(* CODESYS project 车床桁架_RECOVERED_2024-04-15T14-33-14.project
   CompiledLibraryCompatibilityVersion: LeadSysStudio V3.5 SP15 Patch 4
   Title: 车床桁架

Project tree, tasks and I/O mapping:
  Device : SC5-C0A4, Leadshine Technology Co., Ltd., order no. 504001, version 3.5.15.40
    application Application
      libraries: Standard, * (System)
      task MainTask (cyclic, interval t#20ms, priority 1) calls PLC_PRG, 气缸, Public_Prog, OP1001, OP1002
      task EtherCAT_Master_Leadshine_A (cyclic, interval 4000 µs, priority 0) calls EtherCAT_Master_Leadshine_A.EtherCAT_Task, Servo_Ctrol
      program 回原 [LD]
      FunctionBlock/
        function block FB102_ClockPuls [LD]
        program Public_Prog [LD]: SystemVar
        function block FB_CylinderDouble [ST]
        function block FB_CylinderSingle [ST]
      global variables HMI
      global variables I_List
      global variables Alarm
      Symbols
      data type CYLINDER_REF
      global variables 气缸_STRUCT
      program OP1002 [LD]: 辅助流程
      global variables System
      program 气缸 [LD]
      program Servo_Ctrol [LD]
      global variables Publics
      interface ITF
      global variables PersistentVars
      program PLC_PRG [LD]
      program OP1001 [LD]
      global variables O_Lisk
    Device Diagnose
    Network Configuration
      LocalBus Config
    Resource Usage
    LocalBus_Master_Module : LocalBusR1 Master, Leadshine Technology Co., Ltd., version 3.5.15.40
      SC0032N1 : SC0032N1, Leadshine Technology Co., Ltd., version 3.5.15.40
          settings: 位置号 = 1
          unmapped channels: OUTPUT_0, OUTPUT_1, OUTPUT_2, OUTPUT_3
      SC3200 : SC3200, Leadshine Technology Co., Ltd., version 3.5.15.40
          settings: 位置号 = 0
          unmapped channels: INPUT_0, INPUT_1, INPUT_2, INPUT_3
    Modbus_Slave_RS232_COM : Modbus Slave RS232 COM, Leadshine Technology Co., Ltd., version 3.5.15.40
        settings: Vendor.Baudrate = 115200
    SoftMotion General Axis Pool
    EtherCAT_Master_Leadshine_A : EtherCAT Master SoftMotion, 3S - Smart Software Solutions GmbH, version 3.5.16.30
        settings: NetworkName = 'ecat'; SelectNetworkByName = TRUE
      L6N_2 : L6N(COE), Leadshine Technology Co.,Ltd., order no. L6N, version Revision=16#00000001
          settings: DC sync0 cycletime = 4000; DC sync1 cycletime = 4000; Number of SDO = 6; Homing method.Index = 16#6098; Homing method.Subindex = 16#00; Homing method.Value = 35; Homing method.Size = 8; Homing method.AbortIfError = FALSE; Homing method.JumpToLine = FALSE; Homing method.Line = 0; Homing method.CompleteAccess = FALSE; Homing velocity (fast).Index = 16#6099; Homing velocity (fast).Subindex = 16#01; Homing velocity (fast).Value = 6103261; Homing velocity (fast).Size = 32; Homing velocity (fast).AbortIfError = FALSE; Homing velocity (fast).JumpToLine = FALSE; Homing velocity (fast).Line = 0; Homing velocity (fast).CompleteAccess = FALSE; Homing velocity (slow).Index = 16#6099; Homing velocity (slow).Subindex = 16#02; Homing velocity (slow).Value = 1220652; Homing velocity (slow).Size = 32; Homing velocity (slow).AbortIfError = FALSE; Homing velocity (slow).JumpToLine = FALSE; Homing velocity (slow).Line = 0; Homing velocity (slow).CompleteAccess = FALSE; Homing acceleration.Index = 16#609A; Homing acceleration.Subindex = 16#00; Homing acceleration.Value = 61032615; Homing acceleration.Size = 32; Homing acceleration.AbortIfError = FALSE; Homing acceleration.JumpToLine = FALSE; Homing acceleration.Line = 0; Homing acceleration.CompleteAccess = FALSE; Homing offset.Index = 16#607C; Homing offset.Subindex = 16#00; Homing offset.Value = 0; Homing offset.Size = 32; Homing offset.AbortIfError = FALSE;
            Homing offset.JumpToLine = FALSE; Homing offset.Line = 0; Homing offset.CompleteAccess = FALSE
          unmapped channels: Control word, Profile target position, Touch Probe Function, Last error code, Status word, Modes of operation display, Position loop error, Actual motor torque, Actual motor position, Touch Probe Status, Touch probe pos1 pos value, Digital inputs
        Axis_2 : Axis, 3S - Smart Software Solutions GmbH, order no. 0, version 4.6.1.0
            settings: wDriveID = 2; bVirtual = TRUE; dwRatioTechUnitsDenom = 610326149; iRatioTechUnitsNum = 1000; fSWMaxVelocity = 1000; fSWMaxAcceleration = 10000; fSWMaxDeceleration = 10000; fSWMaxJerk = 100000; 一圈脉冲数 = 8388608; 工作台一圈的位移 = 109.955741; 电子齿轮比分子 = 8; 电子齿轮比分母 = 1; ScalingIncs = 8388608; ScalingMotorTurns2 = 8; AdrOffset_8010 = 28; BitOffset_8010 = 0; BitLength_8010 = 16; Address_8010 = '%QW14'; Type_8010 = 'UINT'; AddressPointer_8010 = ADR(%QW14); AdrOffset_8020 = 32; BitOffset_8020 = 0; BitLength_8020 = 32; Address_8020 = '%QD8'; Type_8020 = 'DINT'; AddressPointer_8020 = ADR(%QD8); AdrOffset_8030 = 4294967295; BitOffset_8030 = 0; BitLength_8030 = 32; Address_8030 = ''; Type_8030 = 'DINT'; AddressPointer_8030 = 0; AdrOffset_8040 = 4294967295; BitOffset_8040 = 0; BitLength_8040 = 16; Address_8040 = ''; Type_8040 = 'INT'; AddressPointer_8040 = 0; AdrOffset_8050 = 4294967295; BitOffset_8050 = 0;
              BitLength_8050 = 8; Address_8050 = ''; Type_8050 = 'SINT'; AddressPointer_8050 = 0; AdrOffset_8060 = 36; BitOffset_8060 = 0; BitLength_8060 = 16; Address_8060 = '%QW18'; Type_8060 = 'UINT'; AddressPointer_8060 = ADR(%QW18); AdrOffset_8070 = 4294967295; BitOffset_8070 = 0; BitLength_8070 = 0; Address_8070 = ''; Type_8070 = ''; AddressPointer_8070 = 0; AdrOffset_8080 = 4294967295; BitOffset_8080 = 0; BitLength_8080 = 16; Address_8080 = ''; Type_8080 = 'INT'; AddressPointer_8080 = 0; AdrOffset_8090 = 4294967295; BitOffset_8090 = 0; BitLength_8090 = 0; Address_8090 = ''; Type_8090 = ''; AddressPointer_8090 = 0; AdrOffset_8510 = 70; BitOffset_8510 = 0; BitLength_8510 = 16; Address_8510 = '%IW35'; Type_8510 = 'UINT'; AddressPointer_8510 = ADR(%IW35); AdrOffset_8520 = 84; BitOffset_8520 = 0; BitLength_8520 = 32; Address_8520 = '%ID21'; Type_8520 = 'DINT'; AddressPointer_8520 = ADR(%ID21);
              AdrOffset_8530 = 4294967295; BitOffset_8530 = 0; BitLength_8530 = 0; Address_8530 = ''; Type_8530 = ''; AddressPointer_8530 = 0; AdrOffset_8540 = 80; BitOffset_8540 = 0; BitLength_8540 = 16; Address_8540 = '%IW40'; Type_8540 = 'INT'; AddressPointer_8540 = ADR(%IW40); AdrOffset_8550 = 72; BitOffset_8550 = 0; BitLength_8550 = 8; Address_8550 = '%IB72'; Type_8550 = 'SINT'; AddressPointer_8550 = ADR(%IB72); AdrOffset_8560 = 96; BitOffset_8560 = 0; BitLength_8560 = 32; Address_8560 = '%ID24'; Type_8560 = 'UDINT'; AddressPointer_8560 = ADR(%ID24); AdrOffset_8570 = 88; BitOffset_8570 = 0; BitLength_8570 = 16; Address_8570 = '%IW44'; Type_8570 = 'UINT'; AddressPointer_8570 = ADR(%IW44); AdrOffset_8580 = 92; BitOffset_8580 = 0; BitLength_8580 = 32; Address_8580 = '%ID23'; Type_8580 = 'DINT'; AddressPointer_8580 = ADR(%ID23); AdrOffset_8590 = 4294967295; BitOffset_8590 = 0; BitLength_8590 = 0; Address_8590 = '';
              Type_8590 = ''; AddressPointer_8590 = 0; AdrOffset_8600 = 4294967295; BitOffset_8600 = 0; BitLength_8600 = 0; Address_8600 = ''; Type_8600 = ''; AddressPointer_8600 = 0; AdrOffset_8600 = 4294967295; BitOffset_8600 = 0; BitLength_8600 = 0; Address_8610 = ''; Type_8610 = ''; AddressPointer_8610 = 0; AdrOffset_8620 = 76; BitOffset_8620 = 0; BitLength_8620 = 32; Address_8620 = '%ID19'; Type_8620 = 'DINT'; AddressPointer_8620 = ADR(%ID19)
      L6N_3 : L6N(COE), Leadshine Technology Co.,Ltd., order no. L6N, version Revision=16#00000001
          settings: DC sync0 cycletime = 4000; DC sync1 cycletime = 4000; Number of SDO = 6; Homing method.Index = 16#6098; Homing method.Subindex = 16#00; Homing method.Value = 35; Homing method.Size = 8; Homing method.AbortIfError = FALSE; Homing method.JumpToLine = FALSE; Homing method.Line = 0; Homing method.CompleteAccess = FALSE; Homing velocity (fast).Index = 16#6099; Homing velocity (fast).Subindex = 16#01; Homing velocity (fast).Value = 26701769; Homing velocity (fast).Size = 32; Homing velocity (fast).AbortIfError = FALSE; Homing velocity (fast).JumpToLine = FALSE; Homing velocity (fast).Line = 0; Homing velocity (fast).CompleteAccess = FALSE; Homing velocity (slow).Index = 16#6099; Homing velocity (slow).Subindex = 16#02; Homing velocity (slow).Value = 5340354; Homing velocity (slow).Size = 32; Homing velocity (slow).AbortIfError = FALSE; Homing velocity (slow).JumpToLine = FALSE; Homing velocity (slow).Line = 0; Homing velocity (slow).CompleteAccess = FALSE; Homing acceleration.Index = 16#609A; Homing acceleration.Subindex = 16#00; Homing acceleration.Value = 267017690; Homing acceleration.Size = 32; Homing acceleration.AbortIfError = FALSE; Homing acceleration.JumpToLine = FALSE; Homing acceleration.Line = 0; Homing acceleration.CompleteAccess = FALSE; Homing offset.Index = 16#607C; Homing offset.Subindex = 16#00; Homing offset.Value = 0; Homing offset.Size = 32; Homing offset.AbortIfError = FALSE;
            Homing offset.JumpToLine = FALSE; Homing offset.Line = 0; Homing offset.CompleteAccess = FALSE
          unmapped channels: Control word, Profile target position, Touch Probe Function, Last error code, Status word, Modes of operation display, Position loop error, Actual motor torque, Actual motor position, Touch Probe Status, Touch probe pos1 pos value, Digital inputs
        Axis_3 : Axis, 3S - Smart Software Solutions GmbH, order no. 0, version 4.6.1.0
            settings: wDriveID = 3; bVirtual = TRUE; dwRatioTechUnitsDenom = 26701769; iRatioTechUnitsNum = 10; fSWMaxVelocity = 1000; fSWMaxAcceleration = 10000; fSWMaxDeceleration = 10000; fSWMaxJerk = 100000; 一圈脉冲数 = 8388608; 工作台一圈的位移 = 109.955741; 电子齿轮比分子 = 35; 电子齿轮比分母 = 1; ScalingIncs = 8388608; ScalingMotorTurns2 = 35; AdrOffset_8010 = 40; BitOffset_8010 = 0; BitLength_8010 = 16; Address_8010 = '%QW20'; Type_8010 = 'UINT'; AddressPointer_8010 = ADR(%QW20); AdrOffset_8020 = 44; BitOffset_8020 = 0; BitLength_8020 = 32; Address_8020 = '%QD11'; Type_8020 = 'DINT'; AddressPointer_8020 = ADR(%QD11); AdrOffset_8030 = 4294967295; BitOffset_8030 = 0; BitLength_8030 = 32; Address_8030 = ''; Type_8030 = 'DINT'; AddressPointer_8030 = 0; AdrOffset_8040 = 4294967295; BitOffset_8040 = 0; BitLength_8040 = 16; Address_8040 = ''; Type_8040 = 'INT'; AddressPointer_8040 = 0; AdrOffset_8050 = 4294967295; BitOffset_8050 = 0;
              BitLength_8050 = 8; Address_8050 = ''; Type_8050 = 'SINT'; AddressPointer_8050 = 0; AdrOffset_8060 = 48; BitOffset_8060 = 0; BitLength_8060 = 16; Address_8060 = '%QW24'; Type_8060 = 'UINT'; AddressPointer_8060 = ADR(%QW24); AdrOffset_8070 = 4294967295; BitOffset_8070 = 0; BitLength_8070 = 0; Address_8070 = ''; Type_8070 = ''; AddressPointer_8070 = 0; AdrOffset_8080 = 4294967295; BitOffset_8080 = 0; BitLength_8080 = 16; Address_8080 = ''; Type_8080 = 'INT'; AddressPointer_8080 = 0; AdrOffset_8090 = 4294967295; BitOffset_8090 = 0; BitLength_8090 = 0; Address_8090 = ''; Type_8090 = ''; AddressPointer_8090 = 0; AdrOffset_8510 = 102; BitOffset_8510 = 0; BitLength_8510 = 16; Address_8510 = '%IW51'; Type_8510 = 'UINT'; AddressPointer_8510 = ADR(%IW51); AdrOffset_8520 = 116; BitOffset_8520 = 0; BitLength_8520 = 32; Address_8520 = '%ID29'; Type_8520 = 'DINT'; AddressPointer_8520 = ADR(%ID29);
              AdrOffset_8530 = 4294967295; BitOffset_8530 = 0; BitLength_8530 = 0; Address_8530 = ''; Type_8530 = ''; AddressPointer_8530 = 0; AdrOffset_8540 = 112; BitOffset_8540 = 0; BitLength_8540 = 16; Address_8540 = '%IW56'; Type_8540 = 'INT'; AddressPointer_8540 = ADR(%IW56); AdrOffset_8550 = 104; BitOffset_8550 = 0; BitLength_8550 = 8; Address_8550 = '%IB104'; Type_8550 = 'SINT'; AddressPointer_8550 = ADR(%IB104); AdrOffset_8560 = 128; BitOffset_8560 = 0; BitLength_8560 = 32; Address_8560 = '%ID32'; Type_8560 = 'UDINT'; AddressPointer_8560 = ADR(%ID32); AdrOffset_8570 = 120; BitOffset_8570 = 0; BitLength_8570 = 16; Address_8570 = '%IW60'; Type_8570 = 'UINT'; AddressPointer_8570 = ADR(%IW60); AdrOffset_8580 = 124; BitOffset_8580 = 0; BitLength_8580 = 32; Address_8580 = '%ID31'; Type_8580 = 'DINT'; AddressPointer_8580 = ADR(%ID31); AdrOffset_8590 = 4294967295; BitOffset_8590 = 0; BitLength_8590 = 0; Address_8590 = '';
              Type_8590 = ''; AddressPointer_8590 = 0; AdrOffset_8600 = 4294967295; BitOffset_8600 = 0; BitLength_8600 = 0; Address_8600 = ''; Type_8600 = ''; AddressPointer_8600 = 0; AdrOffset_8600 = 4294967295; BitOffset_8600 = 0; BitLength_8600 = 0; Address_8610 = ''; Type_8610 = ''; AddressPointer_8610 = 0; AdrOffset_8620 = 108; BitOffset_8620 = 0; BitLength_8620 = 32; Address_8620 = '%ID27'; Type_8620 = 'DINT'; AddressPointer_8620 = ADR(%ID27)
      L6N_1 : L6N(COE), Leadshine Technology Co.,Ltd., order no. L6N, version Revision=16#00000001
          settings: DC sync0 cycletime = 4000; DC sync1 cycletime = 4000; Number of SDO = 6; Homing method.Index = 16#6098; Homing method.Subindex = 16#00; Homing method.Value = 35; Homing method.Size = 8; Homing method.AbortIfError = FALSE; Homing method.JumpToLine = FALSE; Homing method.Line = 0; Homing method.CompleteAccess = FALSE; Homing velocity (fast).Index = 16#6099; Homing velocity (fast).Subindex = 16#01; Homing velocity (fast).Value = 16777216; Homing velocity (fast).Size = 32; Homing velocity (fast).AbortIfError = FALSE; Homing velocity (fast).JumpToLine = FALSE; Homing velocity (fast).Line = 0; Homing velocity (fast).CompleteAccess = FALSE; Homing velocity (slow).Index = 16#6099; Homing velocity (slow).Subindex = 16#02; Homing velocity (slow).Value = 3355443; Homing velocity (slow).Size = 32; Homing velocity (slow).AbortIfError = FALSE; Homing velocity (slow).JumpToLine = FALSE; Homing velocity (slow).Line = 0; Homing velocity (slow).CompleteAccess = FALSE; Homing acceleration.Index = 16#609A; Homing acceleration.Subindex = 16#00; Homing acceleration.Value = 167772160; Homing acceleration.Size = 32; Homing acceleration.AbortIfError = FALSE; Homing acceleration.JumpToLine = FALSE; Homing acceleration.Line = 0; Homing acceleration.CompleteAccess = FALSE; Homing offset.Index = 16#607C; Homing offset.Subindex = 16#00; Homing offset.Value = 0; Homing offset.Size = 32; Homing offset.AbortIfError = FALSE;
            Homing offset.JumpToLine = FALSE; Homing offset.Line = 0; Homing offset.CompleteAccess = FALSE
          unmapped channels: Control word, Profile target position, Touch Probe Function, Last error code, Status word, Modes of operation display, Position loop error, Actual motor torque, Actual motor position, Touch Probe Status, Touch probe pos1 pos value, Digital inputs
        Axis_1 : Axis, 3S - Smart Software Solutions GmbH, order no. 0, version 4.6.1.0
            settings: bVirtual = TRUE; dwRatioTechUnitsDenom = 8388608; iRatioTechUnitsNum = 5; fSWMaxVelocity = 1000; fSWMaxAcceleration = 10000; fSWMaxDeceleration = 10000; fSWMaxJerk = 100000; 一圈脉冲数 = 8388608; 工作台一圈的位移 = 5; 电子齿轮比分子 = 1; 电子齿轮比分母 = 1; ScalingIncs = 8388608; AdrOffset_8010 = 16; BitOffset_8010 = 0; BitLength_8010 = 16; Address_8010 = '%QW8'; Type_8010 = 'UINT'; AddressPointer_8010 = ADR(%QW8); AdrOffset_8020 = 20; BitOffset_8020 = 0; BitLength_8020 = 32; Address_8020 = '%QD5'; Type_8020 = 'DINT'; AddressPointer_8020 = ADR(%QD5); AdrOffset_8030 = 4294967295; BitOffset_8030 = 0; BitLength_8030 = 32; Address_8030 = ''; Type_8030 = 'DINT'; AddressPointer_8030 = 0; AdrOffset_8040 = 4294967295; BitOffset_8040 = 0; BitLength_8040 = 16; Address_8040 = ''; Type_8040 = 'INT'; AddressPointer_8040 = 0; AdrOffset_8050 = 4294967295; BitOffset_8050 = 0; BitLength_8050 = 8; Address_8050 = '';
              Type_8050 = 'SINT'; AddressPointer_8050 = 0; AdrOffset_8060 = 24; BitOffset_8060 = 0; BitLength_8060 = 16; Address_8060 = '%QW12'; Type_8060 = 'UINT'; AddressPointer_8060 = ADR(%QW12); AdrOffset_8070 = 4294967295; BitOffset_8070 = 0; BitLength_8070 = 0; Address_8070 = ''; Type_8070 = ''; AddressPointer_8070 = 0; AdrOffset_8080 = 4294967295; BitOffset_8080 = 0; BitLength_8080 = 16; Address_8080 = ''; Type_8080 = 'INT'; AddressPointer_8080 = 0; AdrOffset_8090 = 4294967295; BitOffset_8090 = 0; BitLength_8090 = 0; Address_8090 = ''; Type_8090 = ''; AddressPointer_8090 = 0; AdrOffset_8510 = 38; BitOffset_8510 = 0; BitLength_8510 = 16; Address_8510 = '%IW19'; Type_8510 = 'UINT'; AddressPointer_8510 = ADR(%IW19); AdrOffset_8520 = 52; BitOffset_8520 = 0; BitLength_8520 = 32; Address_8520 = '%ID13'; Type_8520 = 'DINT'; AddressPointer_8520 = ADR(%ID13); AdrOffset_8530 = 4294967295; BitOffset_8530 = 0;
              BitLength_8530 = 0; Address_8530 = ''; Type_8530 = ''; AddressPointer_8530 = 0; AdrOffset_8540 = 48; BitOffset_8540 = 0; BitLength_8540 = 16; Address_8540 = '%IW24'; Type_8540 = 'INT'; AddressPointer_8540 = ADR(%IW24); AdrOffset_8550 = 40; BitOffset_8550 = 0; BitLength_8550 = 8; Address_8550 = '%IB40'; Type_8550 = 'SINT'; AddressPointer_8550 = ADR(%IB40); AdrOffset_8560 = 64; BitOffset_8560 = 0; BitLength_8560 = 32; Address_8560 = '%ID16'; Type_8560 = 'UDINT'; AddressPointer_8560 = ADR(%ID16); AdrOffset_8570 = 56; BitOffset_8570 = 0; BitLength_8570 = 16; Address_8570 = '%IW28'; Type_8570 = 'UINT'; AddressPointer_8570 = ADR(%IW28); AdrOffset_8580 = 60; BitOffset_8580 = 0; BitLength_8580 = 32; Address_8580 = '%ID15'; Type_8580 = 'DINT'; AddressPointer_8580 = ADR(%ID15); AdrOffset_8590 = 4294967295; BitOffset_8590 = 0; BitLength_8590 = 0; Address_8590 = ''; Type_8590 = ''; AddressPointer_8590 = 0;
              AdrOffset_8600 = 4294967295; BitOffset_8600 = 0; BitLength_8600 = 0; Address_8600 = ''; Type_8600 = ''; AddressPointer_8600 = 0; AdrOffset_8600 = 4294967295; BitOffset_8600 = 0; BitLength_8600 = 0; Address_8610 = ''; Type_8610 = ''; AddressPointer_8610 = 0; AdrOffset_8620 = 44; BitOffset_8620 = 0; BitLength_8620 = 32; Address_8620 = '%ID11'; Type_8620 = 'DINT'; AddressPointer_8620 = ADR(%ID11)
      L6N : L6N(COE), Leadshine Technology Co.,Ltd., order no. L6N, version Revision=16#00000001
          settings: DC sync0 cycletime = 4000; DC enable = 1; DC sync0 enable = 1; DC sync0 shift time = 0; DC sync1 cycletime = 4000; DC sync1 enable = 0; DC sync1 factor = 'x 1'; DC sync1 shift time = 0; Number of SDO = 6; Homing method.Index = 16#6098; Homing method.Subindex = 16#00; Homing method.Value = 35; Homing method.Size = 8; Homing method.AbortIfError = FALSE; Homing method.JumpToLine = FALSE; Homing method.Line = 0; Homing method.CompleteAccess = FALSE; Homing velocity (fast).Index = 16#6099; Homing velocity (fast).Subindex = 16#01; Homing velocity (fast).Value = 20971520; Homing velocity (fast).Size = 32; Homing velocity (fast).AbortIfError = FALSE; Homing velocity (fast).JumpToLine = FALSE; Homing velocity (fast).Line = 0; Homing velocity (fast).CompleteAccess = FALSE; Homing velocity (slow).Index = 16#6099; Homing velocity (slow).Subindex = 16#02; Homing velocity (slow).Value = 4194304; Homing velocity (slow).Size = 32; Homing velocity (slow).AbortIfError = FALSE; Homing velocity (slow).JumpToLine = FALSE; Homing velocity (slow).Line = 0; Homing velocity (slow).CompleteAccess = FALSE; Homing acceleration.Index = 16#609A; Homing acceleration.Subindex = 16#00; Homing acceleration.Value = 209715200; Homing acceleration.Size = 32; Homing acceleration.AbortIfError = FALSE; Homing acceleration.JumpToLine = FALSE; Homing acceleration.Line = 0;
            Homing acceleration.CompleteAccess = FALSE; Homing offset.Index = 16#607C; Homing offset.Subindex = 16#00; Homing offset.Value = 0; Homing offset.Size = 32; Homing offset.AbortIfError = FALSE; Homing offset.JumpToLine = FALSE; Homing offset.Line = 0; Homing offset.CompleteAccess = FALSE
          unmapped channels: Control word, Profile target position, Touch Probe Function, Last error code, Status word, Modes of operation display, Position loop error, Actual motor torque, Actual motor position, Touch Probe Status, Touch probe pos1 pos value, Digital inputs
        Axis : Axis, 3S - Smart Software Solutions GmbH, order no. 0, version 4.6.1.0
            settings: wDriveID = 0; bVirtual = TRUE; dwRatioTechUnitsDenom = 2097152; fSWMaxVelocity = 1000; fSWMaxAcceleration = 10000; fSWMaxDeceleration = 10000; fSWMaxJerk = 100000; 一圈脉冲数 = 8388608; 工作台一圈的位移 = 4; 电子齿轮比分子 = 1; 电子齿轮比分母 = 1; ScalingIncs = 8388608; AdrOffset_8010 = 4; BitOffset_8010 = 0; BitLength_8010 = 16; Address_8010 = '%QW2'; Type_8010 = 'UINT'; AddressPointer_8010 = ADR(%QW2); AdrOffset_8020 = 8; BitOffset_8020 = 0; BitLength_8020 = 32; Address_8020 = '%QD2'; Type_8020 = 'DINT'; AddressPointer_8020 = ADR(%QD2); AdrOffset_8030 = 4294967295; BitOffset_8030 = 0; BitLength_8030 = 32; Address_8030 = ''; Type_8030 = 'DINT'; AddressPointer_8030 = 0; AdrOffset_8040 = 4294967295; BitOffset_8040 = 0; BitLength_8040 = 16; Address_8040 = ''; Type_8040 = 'INT'; AddressPointer_8040 = 0; AdrOffset_8050 = 4294967295; BitOffset_8050 = 0; BitLength_8050 = 8; Address_8050 = '';
              Type_8050 = 'SINT'; AddressPointer_8050 = 0; AdrOffset_8060 = 12; BitOffset_8060 = 0; BitLength_8060 = 16; Address_8060 = '%QW6'; Type_8060 = 'UINT'; AddressPointer_8060 = ADR(%QW6); AdrOffset_8070 = 4294967295; BitOffset_8070 = 0; BitLength_8070 = 0; Address_8070 = ''; Type_8070 = ''; AddressPointer_8070 = 0; AdrOffset_8080 = 4294967295; BitOffset_8080 = 0; BitLength_8080 = 16; Address_8080 = ''; Type_8080 = 'INT'; AddressPointer_8080 = 0; AdrOffset_8090 = 4294967295; BitOffset_8090 = 0; BitLength_8090 = 0; Address_8090 = ''; Type_8090 = ''; AddressPointer_8090 = 0; AdrOffset_8510 = 6; BitOffset_8510 = 0; BitLength_8510 = 16; Address_8510 = '%IW3'; Type_8510 = 'UINT'; AddressPointer_8510 = ADR(%IW3); AdrOffset_8520 = 20; BitOffset_8520 = 0; BitLength_8520 = 32; Address_8520 = '%ID5'; Type_8520 = 'DINT'; AddressPointer_8520 = ADR(%ID5); AdrOffset_8530 = 4294967295; BitOffset_8530 = 0;
              BitLength_8530 = 0; Address_8530 = ''; Type_8530 = ''; AddressPointer_8530 = 0; AdrOffset_8540 = 16; BitOffset_8540 = 0; BitLength_8540 = 16; Address_8540 = '%IW8'; Type_8540 = 'INT'; AddressPointer_8540 = ADR(%IW8); AdrOffset_8550 = 8; BitOffset_8550 = 0; BitLength_8550 = 8; Address_8550 = '%IB8'; Type_8550 = 'SINT'; AddressPointer_8550 = ADR(%IB8); AdrOffset_8560 = 32; BitOffset_8560 = 0; BitLength_8560 = 32; Address_8560 = '%ID8'; Type_8560 = 'UDINT'; AddressPointer_8560 = ADR(%ID8); AdrOffset_8570 = 24; BitOffset_8570 = 0; BitLength_8570 = 16; Address_8570 = '%IW12'; Type_8570 = 'UINT'; AddressPointer_8570 = ADR(%IW12); AdrOffset_8580 = 28; BitOffset_8580 = 0; BitLength_8580 = 32; Address_8580 = '%ID7'; Type_8580 = 'DINT'; AddressPointer_8580 = ADR(%ID7); AdrOffset_8590 = 4294967295; BitOffset_8590 = 0; BitLength_8590 = 0; Address_8590 = ''; Type_8590 = ''; AddressPointer_8590 = 0;
              AdrOffset_8600 = 4294967295; BitOffset_8600 = 0; BitLength_8600 = 0; Address_8600 = ''; Type_8600 = ''; AddressPointer_8600 = 0; AdrOffset_8600 = 4294967295; BitOffset_8600 = 0; BitLength_8600 = 0; Address_8610 = ''; Type_8610 = ''; AddressPointer_8610 = 0; AdrOffset_8620 = 12; BitOffset_8620 = 0; BitLength_8620 = 32; Address_8620 = '%ID3'; Type_8620 = 'DINT'; AddressPointer_8620 = ADR(%ID3)
*)

// Device/Application/CYLINDER_REF
TYPE CYLINDER_REF :
STRUCT
	///初始化时返回原位控制
	xInit: BOOL;
	///自动控制,变为TRUE时，执行到位控制，变为FALSE时执行原位控制
	xAutoCmd: BOOL;
	///到位标志,处于原位状态
	xIsBack: BOOL;
	///到位标志,处于到位状态	
	xIsFront: BOOL;
END_STRUCT
END_TYPE

// Device/Application/HMI
{attribute 'qualified_only'}
VAR_GLOBAL
END_VAR
VAR_GLOBAL
	报警复位 AT %MX0.0: BOOL;
END_VAR
VAR_GLOBAL RETAIN PERSISTENT
	上料推出气缸原位延时 AT %MW1002: WORD := 10;
	上料推出气缸到位延时 AT %MW1003: WORD := 10;
END_VAR
VAR_GLOBAL
	上料顶起气缸_ON_UP AT %MX0.3: BOOL;
END_VAR
VAR_GLOBAL RETAIN PERSISTENT
	上料顶起气缸原位延时 AT %MW1000: WORD := 10;
	上料顶起气缸到位位延时 AT %MW1001: WORD := 10;
END_VAR
VAR_GLOBAL
	上料气动振动筛_ON_UP AT %MX0.6: BOOL;
	X轴失能 AT %MX0.7: BOOL;
	Z2轴失能 AT %MX1.0: BOOL;
	Z1轴失能 AT %MX1.1: BOOL;
	Y轴失能 AT %MX1.2: BOOL;
	X轴_CCW AT %MX1.3: BOOL;
	X轴_CW AT %MX1.4: BOOL;
	Y轴_CCW AT %MX1.5: BOOL;
	Y轴_CW AT %MX0.5: BOOL;
	Z1轴_CCW AT %MX0.4: BOOL;
	Z1轴_CW AT %MX1.6: BOOL;
	Z2轴_CCW AT %MX0.2: BOOL;
	Z2轴_CW AT %MX0.1: BOOL;
	上料推出气缸_ON_UP AT %MX1.7: BOOL;
END_VAR
VAR_GLOBAL RETAIN PERSISTENT
	X轴手动速度 AT %MD1000: REAL := 20;
	Z1轴手动速度 AT %MD1002: REAL := 20;
	Y轴手动速度 AT %MD1001: REAL := 20;
	Z2轴手动速度 AT %MD1003: REAL := 20;
	X轴手动减速度: REAL := 1000;
	X轴手动加速度: REAL := 1000;
	Y轴手动加速度: REAL := 1000;
	Y轴手动减速度: REAL := 1000;
	Z1轴手动减速度: REAL := 1000;
	Z1轴手动加速度: REAL := 1000;
	Z2轴手动减速度: REAL := 1000;
	Z2轴手动加速度: REAL := 1000;
END_VAR
VAR_GLOBAL
	X轴错误代码: DWORD;
	X状态_未使能 AT %MX2.4: BOOL;
	X状态_报错 AT %MX2.5: BOOL;
	X状态_停止中 AT %MX2.6: BOOL;
	X状态_准备好 AT %MX2.7: BOOL;
	X状态_点位运动 AT %MX3.0: BOOL;
	X状态_连续运动: BOOL;
	X状态_同步运动: BOOL;
	X状态_回零中: BOOL;
	X状态_恒速运动 AT %MX3.1: BOOL;
	X状态_加速中 AT %MX3.2: BOOL;
	X状态_减速中 AT %MX3.3: BOOL;
	X状态_超过软限制 AT %MX3.4: BOOL;
	Y轴错误代码: DWORD;
	Y状态_未使能 AT %MX3.5: BOOL;
	Y状态_报错 AT %MX3.6: BOOL;
	Y状态_停止中 AT %MX3.7: BOOL;
	Y状态_准备好 AT %MX4.0: BOOL;
	Y状态_点位运动 AT %MX4.1: BOOL;
	Y状态_连续运动: BOOL;
	Y状态_同步运动: BOOL;
	Y状态_回零中: BOOL;
	Y状态_恒速运动 AT %MX4.2: BOOL;
	Y状态_加速中 AT %MX4.3: BOOL;
	Y状态_减速中 AT %MX4.4: BOOL;
	Y状态_超过软限制 AT %MX4.5: BOOL;
	Z1轴错误代码: DWORD;
	Z1状态_未使能 AT %MX4.6: BOOL;
	Z1状态_报错 AT %MX4.7: BOOL;
	Z1状态_停止中 AT %MX5.0: BOOL;
	Z1状态_准备好 AT %MX5.1: BOOL;
	Z1状态_点位运动 AT %MX5.2: BOOL;
	Z1状态_连续运动: BOOL;
	Z1状态_同步运动: BOOL;
	Z1状态_回零中: BOOL;
	Z1状态_恒速运动 AT %MX5.3: BOOL;
	Z1状态_加速中 AT %MX5.4: BOOL;
	Z1状态_减速中 AT %MX5.5: BOOL;
	Z1状态_超过软限制 AT %MX5.6: BOOL;
	Z2轴错误代码: DWORD;
	Z2状态_未使能 AT %MX5.7: BOOL;
	Z2状态_报错 AT %mx6.0: BOOL;
	Z2状态_停止中 AT %mx6.1: BOOL;
	Z2状态_准备好 AT %MX6.7: BOOL;
	Z2状态_点位运动 AT %MX6.2: BOOL;
	Z2状态_连续运动: BOOL;
	Z2状态_同步运动: BOOL;
	Z2状态_回零中: BOOL;
	Z2状态_恒速运动 AT %MX6.3: BOOL;
	Z2状态_加速中 AT %MX6.4: BOOL;
	Z2状态_减速中 AT %MX6.5: BOOL;
	Z2状态_超过软限制 AT %MX6.6: BOOL;
	上料气爪_ON_UP AT %MX2.3: BOOL;
	开门气缸_ON_UP AT %MX2.2: BOOL;
	翻转气缸_ON_UP AT %MX2.1: BOOL;
	下料气爪_ON_UP AT %MX2.0: BOOL;
END_VAR
VAR_GLOBAL RETAIN PERSISTENT
	点位P0 AT %MD2000: ARRAY[0..3] OF REAL;
	点位P1 AT %MD2004: ARRAY[0..3] OF REAL;
END_VAR

VAR_GLOBAL
	Y轴当前位置 AT %MD1005: REAL;
	Z2轴当前位置 AT %MD1007: REAL;
	Z1轴当前位置 AT %MD1006: REAL;
	X轴当前位置 AT %MD1004: REAL;
	Z2当前速度: REAL;
	Z1当前速度: REAL;
	Y轴当前速度: REAL;
	X轴当前速度: REAL;
END_VAR
VAR_GLOBAL RETAIN PERSISTENT
	上料气爪原位延时 AT %MW1004: WORD := 10;
	上料气爪到位延时 AT %MW1005: WORD := 10;
	下料气爪到位延时 AT %MW1006: WORD := 10;
	下料气爪原位延时 AT %MW1007: WORD := 10;
	翻转气爪到位延时 AT %MW1008: WORD := 10;
	翻转气爪原位延时 AT %MW1009: WORD := 10;
	开门气缸原位延时 AT %MW1010: WORD := 50;
	开门气缸到位延时 AT %MW1011: WORD := 50;
	点位P9 AT %MD2036: ARRAY[0..3] OF REAL;
	点位P8 AT %MD2032: ARRAY[0..3] OF REAL;
	点位P7 AT %MD2028: ARRAY[0..3] OF REAL;
	点位P6 AT %MD2024: ARRAY[0..3] OF REAL;
	点位P5 AT %MD2020: ARRAY[0..3] OF REAL;
	点位P4 AT %MD2016: ARRAY[0..3] OF REAL;
	点位P3 AT %MD2012: ARRAY[0..3] OF REAL;
	点位P2 AT %MD2008: ARRAY[0..3] OF REAL;
	点位P10 AT %MD2040: ARRAY[0..3] OF REAL;
END_VAR

// Device/Application/I_List
{attribute 'qualified_only'}
VAR_GLOBAL
	// 上料传送带到位确认
	X0 AT %IX0.0: BOOL;
	// 紧急停止
	X1 AT %IX0.1: BOOL;
	// 推出气缸原位
	X2 AT %IX0.2: BOOL;
	// 推出气缸动作位
	X3 AT %IX0.3: BOOL;
	// 顶起气缸原位
	X4 AT %IX0.4: BOOL;
	// 顶起气缸动作位
	X5 AT %IX0.5: BOOL;
	// 上料气爪原位
	X6 AT %IX0.6: BOOL;
	// 上料气爪动作位
	X7 AT %IX0.7: BOOL;
	// 下料气爪原位
	X10 AT %IX1.0: BOOL;
	// 下料气爪动作位
	X11 AT %IX1.1: BOOL;
	// 翻转气缸原位
	X12 AT %IX1.2: BOOL;
	// 翻转气缸动作位
	X13 AT %IX1.3: BOOL;
	// 开门气缸原位
	X14 AT %IX1.4: BOOL;
	// 开门气缸动作位
	X15 AT %IX1.5: BOOL;
	// 启动按钮
	X16 AT %IX1.6: BOOL;
	// 停止按钮
	X17 AT %IX1.7: BOOL;
	// 复位按钮
	X20 AT %IX2.0: BOOL;
	// 手自动按钮ON为自动
	X21 AT %IX2.1: BOOL;
	// 下料确认
	X22 AT %IX2.2: BOOL;
	// 联机卡盘夹紧
	X23 AT %IX2.3: BOOL;
	// 联机启动
	X24 AT %IX2.4: BOOL;
	// 联机停止
	X25 AT %IX2.5: BOOL;
	// 联机故障
	X26 AT %IX2.6: BOOL;
	// 联机X轴零点
	X27 AT %IX2.7: BOOL;
	// 联机Z轴零点
	X30 AT %IX3.0: BOOL;
	X31 AT %IX3.1: BOOL;
	X32 AT %IX3.2: BOOL;
	X33 AT %IX3.3: BOOL;
	X34 AT %IX3.4: BOOL;
	X35 AT %IX3.5: BOOL;
	X36 AT %IX3.6: BOOL;
	X37 AT %IX3.7: BOOL;
END_VAR

// Device/Application/Alarm
{attribute 'qualified_only'}
VAR_GLOBAL
END_VAR
VAR_GLOBAL
	设备急停 AT %MX100.0: BOOL;
	推出气缸手自动不一致报警 AT %MX100.1: BOOL;
	推出气缸原位报警 AT %MX100.2: BOOL;
	推出气缸到位报警 AT %MX100.3: BOOL;
	顶起气缸手自动不一致报警 AT %MX100.4: BOOL;
	顶起气缸原位报警 AT %MX100.5: BOOL;
	顶起气缸到位报警 AT %MX100.6: BOOL;
	上料气爪手自动不一致报警 AT %MX100.7: BOOL;
	上料气爪原位报警 AT %MX101.0: BOOL;
	上料气爪到位报警 AT %MX101.1: BOOL;
	下料气爪手自动不一致报警 AT %MX101.2: BOOL;
	下料气爪原位报警 AT %MX101.3: BOOL;
	下料气爪到位报警 AT %MX101.4: BOOL;
	翻转气缸手自动不一致报警 AT %MX101.5: BOOL;
	翻转气缸原位报警 AT %MX101.6: BOOL;
	翻转气缸到位报警 AT %MX101.7: BOOL;
	开门气缸手自动不一致报警 AT %MX102.0: BOOL;
	开门气缸原位报警 AT %MX102.1: BOOL;
	开门气缸到位报警 AT %MX102.2: BOOL;
END_VAR

// Device/Application/气缸_STRUCT
{attribute 'qualified_only'}
VAR_GLOBAL
	上料推出气缸: CYLINDER_REF;
	上料顶起气缸: CYLINDER_REF;
	上料振动筛: CYLINDER_REF;
	开门气缸: CYLINDER_REF;
	翻转气缸: CYLINDER_REF;
	上料气爪: CYLINDER_REF;
	下料气爪: CYLINDER_REF;
END_VAR

// Device/Application/System
{attribute 'qualified_only'}
VAR_GLOBAL
	// 上电扫描一周期
FirstScan    :BOOL;
// 常ON
AlwaysTRUE   : BOOL;
// 常OFF
AlwaysFALSE  : BOOL;
// 0.1S周期脉冲
Clock_10Hz    :BOOL;
// 0.2S周期脉冲
Clock_5Hz    :BOOL;
// 0.5S周期脉冲
Clock_2Hz    :BOOL;
// 1S周期脉冲
Clock_1Hz    :BOOL;
// 2S周期脉冲
Clock_HalfHz :BOOL;
END_VAR

// Device/Application/Publics
{attribute 'qualified_only'}
VAR_GLOBAL
	// 调试使用常ON
CYGIA_ON   :BOOL;
// 调试使用常OFF
CYGIA_OFF  :BOOL;
	启动上升: BOOL;
	警报: BOOL;
	暂停: BOOL;
	EMG: BOOL;
	X定位数据: REAL;
	Y定位数据: REAL;
	Z1定位数据: REAL;
	Z2定位数据: REAL;
	Z2加速度: REAL;
	Z1加速度: REAL;
END_VAR
VAR_GLOBAL RETAIN PERSISTENT
	Y加速度: REAL;
	X加速度: REAL;
	Z2减速度: REAL;
	Z1减速度: REAL;
	Y减速度: REAL;
	X减速度: REAL;
	Z2自动速度: REAL;
	Z1自动速度: REAL;
	Y自动速度: REAL;
	X自动速度: REAL;
END_VAR
VAR_GLOBAL
	Z2轴完成: BOOL;
	Z1轴完成: BOOL;
	Y轴完成: BOOL;
	X轴完成: BOOL;
	Z2轴启动: BOOL;
	Z1轴启动: BOOL;
	Y轴启动: BOOL;
	X轴启动: BOOL;
END_VAR

// Device/Application/PersistentVars
{attribute 'qualified_only'}
VAR_GLOBAL PERSISTENT RETAIN
	// 生成持久变量的实例路径
	HMI.上料推出气缸原位延时: WORD := WORD#10;
	// 生成持久变量的实例路径
	HMI.上料推出气缸到位延时: WORD := WORD#10;
	// 生成持久变量的实例路径
	HMI.上料顶起气缸原位延时: WORD := WORD#10;
	// 生成持久变量的实例路径
	HMI.上料顶起气缸到位位延时: WORD := WORD#10;
	// 生成持久变量的实例路径
	HMI.X轴手动速度: REAL := 20.0;
	// 生成持久变量的实例路径
	HMI.Z1轴手动速度: REAL := 20.0;
	// 生成持久变量的实例路径
	HMI.Y轴手动速度: REAL := 20.0;
	// 生成持久变量的实例路径
	HMI.Z2轴手动速度: REAL := 20.0;
	// 生成持久变量的实例路径
	HMI.X轴手动减速度: REAL := 1000.0;
	// 生成持久变量的实例路径
	HMI.X轴手动加速度: REAL := 1000.0;
	// 生成持久变量的实例路径
	HMI.Y轴手动加速度: REAL := 1000.0;
	// 生成持久变量的实例路径
	HMI.Y轴手动减速度: REAL := 1000.0;
	// 生成持久变量的实例路径
	HMI.Z1轴手动减速度: REAL := 1000.0;
	// 生成持久变量的实例路径
	HMI.Z1轴手动加速度: REAL := 1000.0;
	// 生成持久变量的实例路径
	HMI.Z2轴手动减速度: REAL := 1000.0;
	// 生成持久变量的实例路径
	HMI.Z2轴手动加速度: REAL := 1000.0;
	// 生成持久变量的实例路径
	HMI.点位P1: ARRAY [0..3] OF REAL;
	// 生成持久变量的实例路径
	HMI.点位P0: ARRAY [0..3] OF REAL;
	// 生成持久变量的实例路径
	HMI.点位P9: ARRAY [0..3] OF REAL;
	// 生成持久变量的实例路径
	HMI.点位P8: ARRAY [0..3] OF REAL;
	// 生成持久变量的实例路径
	HMI.点位P7: ARRAY [0..3] OF REAL;
	// 生成持久变量的实例路径
	HMI.点位P6: ARRAY [0..3] OF REAL;
	// 生成持久变量的实例路径
	HMI.点位P5: ARRAY [0..3] OF REAL;
	// 生成持久变量的实例路径
	HMI.点位P4: ARRAY [0..3] OF REAL;
	// 生成持久变量的实例路径
	HMI.点位P3: ARRAY [0..3] OF REAL;
	// 生成持久变量的实例路径
	HMI.点位P2: ARRAY [0..3] OF REAL;
	// 生成持久变量的实例路径
	HMI.点位P10: ARRAY [0..3] OF REAL;
	// 生成持久变量的实例路径
	HMI.上料气爪原位延时: WORD := WORD#10;
	// 生成持久变量的实例路径
	HMI.上料气爪到位延时: WORD := WORD#10;
	// 生成持久变量的实例路径
	HMI.下料气爪到位延时: WORD := WORD#10;
	// 生成持久变量的实例路径
	HMI.下料气爪原位延时: WORD := WORD#10;
	// 生成持久变量的实例路径
	HMI.翻转气爪到位延时: WORD := WORD#10;
	// 生成持久变量的实例路径
	HMI.翻转气爪原位延时: WORD := WORD#10;
	// 生成持久变量的实例路径
	HMI.开门气缸原位延时: WORD := WORD#50;
	// 生成持久变量的实例路径
	HMI.开门气缸到位延时: WORD := WORD#50;
	// 生成持久变量的实例路径
	Publics.Y加速度: REAL;
	// 生成持久变量的实例路径
	Publics.X加速度: REAL;
	// 生成持久变量的实例路径
	Publics.Z2减速度: REAL;
	// 生成持久变量的实例路径
	Publics.Z1减速度: REAL;
	// 生成持久变量的实例路径
	Publics.Y减速度: REAL;
	// 生成持久变量的实例路径
	Publics.X减速度: REAL;
	// 生成持久变量的实例路径
	Publics.Z2自动速度: REAL;
	// 生成持久变量的实例路径
	Publics.Z1自动速度: REAL;
	// 生成持久变量的实例路径
	Publics.Y自动速度: REAL;
	// 生成持久变量的实例路径
	Publics.X自动速度: REAL;
END_VAR

// Device/Application/O_Lisk
{attribute 'qualified_only'}
VAR_GLOBAL
	// 皮带运转
	Y0 AT %QX0.0: BOOL;
	// 震动筛运动
	Y1 AT %QX0.1: BOOL;
	// 推出气缸原位
	Y2 AT %QX0.2: BOOL;
	// 紧急停止输出
	Y3 AT %QX0.3: BOOL;
	// 顶起气缸原位
	Y4 AT %QX0.4: BOOL;
	Y5 AT %QX0.5: BOOL;
	// 上料气爪原位
	Y6 AT %QX0.6: BOOL;
	Y7 AT %QX0.7: BOOL;
	// 下料气爪原位
	Y10 AT %QX1.0: BOOL;
	Y11 AT %QX1.0: BOOL;
	// 翻转气缸原位
	Y12 AT %QX1.0: BOOL;
	Y13 AT %QX1.0: BOOL;
	// 开门气缸原位
	Y14 AT %QX1.0: BOOL;
	Y15 AT %QX1.5: BOOL;
	// 启动按钮LED
	Y16 AT %QX1.6: BOOL;
	// 停止按钮LED
	Y17 AT %QX1.7: BOOL;
	// 复位按钮LED
	Y20 AT %QX2.0: BOOL;
	Y21 AT %QX2.1: BOOL;
	// 下料传送带
	Y22 AT %QX2.2: BOOL;
	// 三色灯红
	Y23 AT %QX2.3: BOOL;
	// 三色灯黄
	Y24 AT %QX2.4: BOOL;
	// 三色灯绿
	Y25 AT %QX2.5: BOOL;
	// 三色灯蜂鸣
	Y26 AT %QX2.6: BOOL;
	// 联机卡盘夹紧
	Y27 AT %QX2.7: BOOL;
	// 联机启动
	Y30 AT %QX3.0: BOOL;
	// 联机停止
	Y31 AT %QX3.1: BOOL;
	Y32 AT %QX3.2: BOOL;
	Y33 AT %QX3.3: BOOL;
	Y34 AT %QX3.4: BOOL;
	Y35 AT %QX3.5: BOOL;
	Y36 AT %QX3.6: BOOL;
	Y37 AT %QX3.7: BOOL;
END_VAR

// Device/Application/PLC_PRG
PROGRAM PLC_PRG
VAR
	SMC3_ReinitDrive_0: SMC3_ReinitDrive;
END_VAR

// NETWORK 1

END_PROGRAM

// Device/Application/气缸
PROGRAM 气缸
VAR
	FB_CylinderSingle_0: FB_CylinderSingle;
	上料推出气缸到位延时: word;
	上料推出气缸原位延时: word;
	FB_CylinderSingle_1: FB_CylinderSingle;
	上料推出气缸报警复位: BOOL;
	上料顶起气缸原位延时: WORD;
	上料顶起气缸到位位延时: WORD;
	FB_CylinderSingle_2: FB_CylinderSingle;
END_VAR

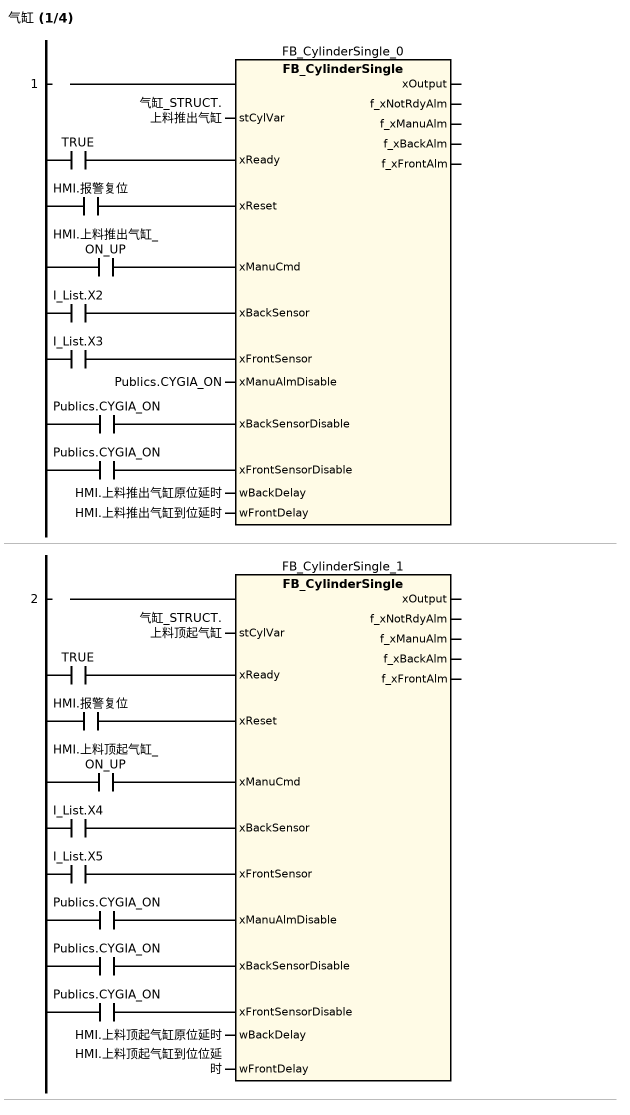
// NETWORK 1
FB_CylinderSingle_0(
    stCylVar := 气缸_STRUCT.上料推出气缸,
    xReady := TRUE,
    xReset := HMI.报警复位,
    xManuCmd := HMI.上料推出气缸_ON_UP,
    xBackSensor := I_List.X2,
    xFrontSensor := I_List.X3,
    xManuAlmDisable := Publics.CYGIA_ON,
    xBackSensorDisable := Publics.CYGIA_ON,
    xFrontSensorDisable := Publics.CYGIA_ON,
    wBackDelay := HMI.上料推出气缸原位延时,
    wFrontDelay := HMI.上料推出气缸到位延时); // FB_CylinderSingle

// NETWORK 2
FB_CylinderSingle_1(
    stCylVar := 气缸_STRUCT.上料顶起气缸,
    xReady := TRUE,
    xReset := HMI.报警复位,
    xManuCmd := HMI.上料顶起气缸_ON_UP,
    xBackSensor := I_List.X4,
    xFrontSensor := I_List.X5,
    xManuAlmDisable := Publics.CYGIA_ON,
    xBackSensorDisable := Publics.CYGIA_ON,
    xFrontSensorDisable := Publics.CYGIA_ON,
    wBackDelay := HMI.上料顶起气缸原位延时,
    wFrontDelay := HMI.上料顶起气缸到位位延时); // FB_CylinderSingle

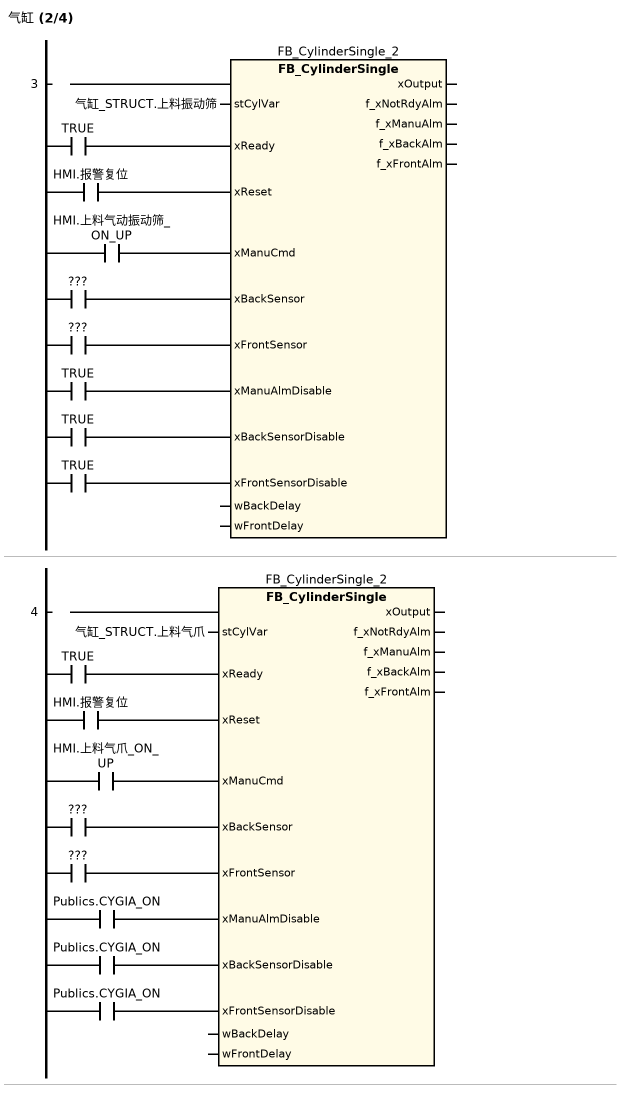
// NETWORK 3
FB_CylinderSingle_2(
    stCylVar := 气缸_STRUCT.上料振动筛,
    xReady := TRUE,
    xReset := HMI.报警复位,
    xManuCmd := HMI.上料气动振动筛_ON_UP,
    xManuAlmDisable := TRUE,
    xBackSensorDisable := TRUE,
    xFrontSensorDisable := TRUE); // FB_CylinderSingle

// NETWORK 4
FB_CylinderSingle_2(
    stCylVar := 气缸_STRUCT.上料气爪,
    xReady := TRUE,
    xReset := HMI.报警复位,
    xManuCmd := HMI.上料气爪_ON_UP,
    xManuAlmDisable := Publics.CYGIA_ON,
    xBackSensorDisable := Publics.CYGIA_ON,
    xFrontSensorDisable := Publics.CYGIA_ON); // FB_CylinderSingle

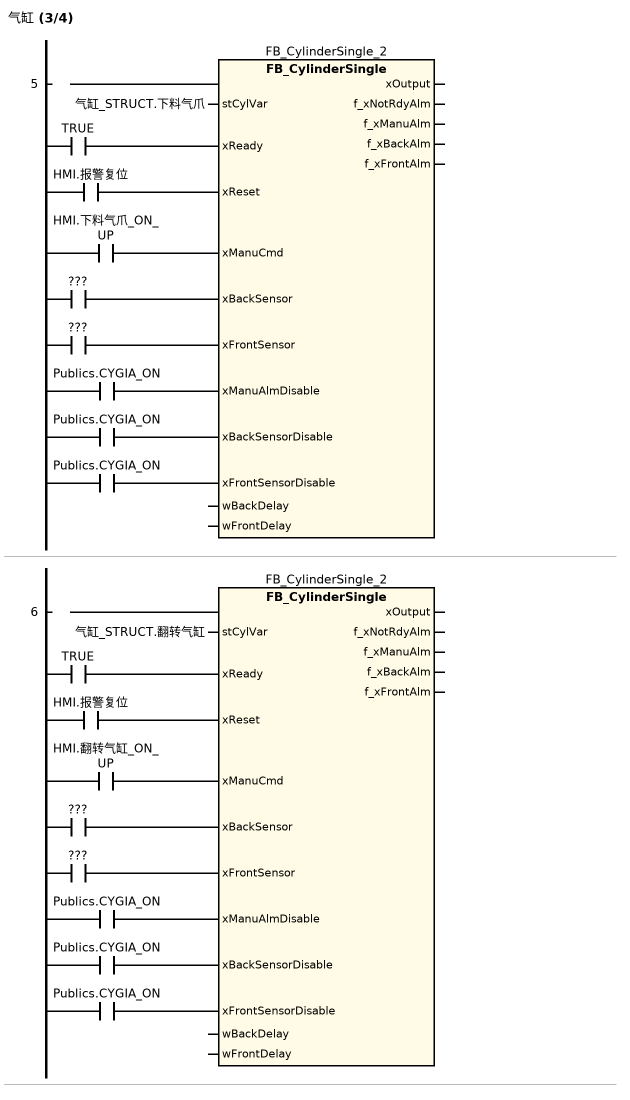
// NETWORK 5
FB_CylinderSingle_2(
    stCylVar := 气缸_STRUCT.下料气爪,
    xReady := TRUE,
    xReset := HMI.报警复位,
    xManuCmd := HMI.下料气爪_ON_UP,
    xManuAlmDisable := Publics.CYGIA_ON,
    xBackSensorDisable := Publics.CYGIA_ON,
    xFrontSensorDisable := Publics.CYGIA_ON); // FB_CylinderSingle

// NETWORK 6
FB_CylinderSingle_2(
    stCylVar := 气缸_STRUCT.翻转气缸,
    xReady := TRUE,
    xReset := HMI.报警复位,
    xManuCmd := HMI.翻转气缸_ON_UP,
    xManuAlmDisable := Publics.CYGIA_ON,
    xBackSensorDisable := Publics.CYGIA_ON,
    xFrontSensorDisable := Publics.CYGIA_ON); // FB_CylinderSingle

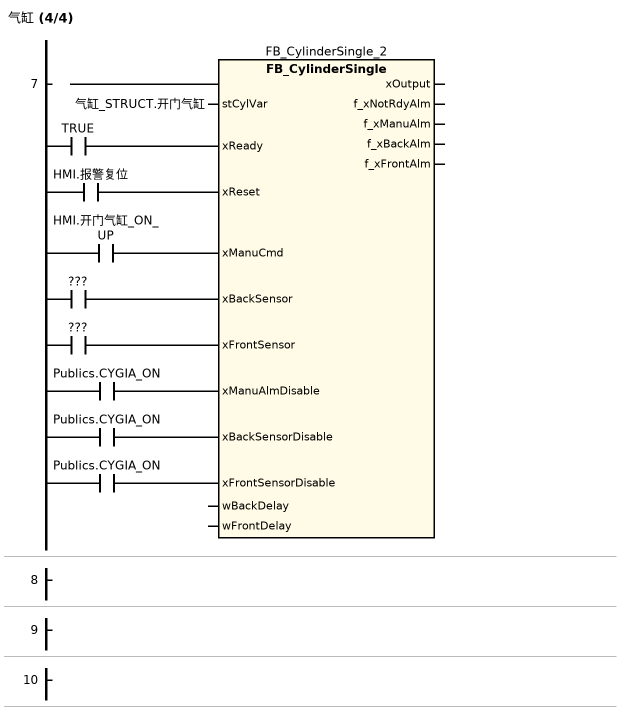
// NETWORK 7
FB_CylinderSingle_2(
    stCylVar := 气缸_STRUCT.开门气缸,
    xReady := TRUE,
    xReset := HMI.报警复位,
    xManuCmd := HMI.开门气缸_ON_UP,
    xManuAlmDisable := Publics.CYGIA_ON,
    xBackSensorDisable := Publics.CYGIA_ON,
    xFrontSensorDisable := Publics.CYGIA_ON); // FB_CylinderSingle

// NETWORK 8

// NETWORK 9

// NETWORK 10

END_PROGRAM

// Device/Application/FunctionBlock/FB_CylinderSingle
FUNCTION_BLOCK FB_CylinderSingle
VAR_IN_OUT
	stCylVar: CYLINDER_REF;
END_VAR
VAR_INPUT
	///安全条件
	xReady: BOOL;
	///报警复位
	xReset: BOOL;
	///手动控制,每on一次,则反转输出点状态
	xManuCmd: BOOL;
	///原位检测
	xBackSensor: BOOL;
	///到位检测
	xFrontSensor: BOOL;
	///手自动不一致报警无效
	xManuAlmDisable: BOOL;
	///原位检测无效
	xBackSensorDisable: BOOL;
	///到位检测无效
	xFrontSensorDisable: BOOL;
	///原位延时
	wBackDelay: WORD;
	///到位延时
	wFrontDelay: WORD;
END_VAR
VAR_OUTPUT
	xOutput: BOOL;
	///未满足安全条件报警
	f_xNotRdyAlm: BOOL;
	///手自动不一致报警	
	f_xManuAlm: BOOL;
	///未在原位报警
	f_xBackAlm: BOOL;
	///未到位报警
	f_xFrontAlm: BOOL;
END_VAR
VAR
	///获取自动控制的上升沿
	fbAutoRise: R_TRIG;
	///获取自动控制的下升沿
	fbAutoFall: F_TRIG;
	///获取手动控制的下升沿
	fbManuFall: F_TRIG;
	///获取复位信号的上升沿
	fbResetRise: R_TRIG;
	///原位状态延时,用于输出原位状态
	fbBackTon: TON;
	///到位状态延时,用于输出到位状态
	fbFrontTon: TON;
	///获取原位状态下降沿	
	fbBackFall: F_TRIG;
	///获取到位状态下降沿
	fbFrontFall: F_TRIG;
	///原位动作超时,用于输出未在原位位置报警
	fbBackWait: TON;
	///到位动作超时,用于输出未在到位位置报警
	fbFrontWait: TON;
END_VAR

   //初始化时复位输出点
   IF xReady AND stCylVar.xInit AND ( NOT f_xNotRdyAlm	) THEN
	    xOutput := FALSE;
	    f_xManuAlm  := FALSE;
	    stCylVar.xInit  := FALSE;
 
   END_IF


   //获取手动控制、自动控制的边沿信号
   fbManuFall(CLK:=xManuCmd , Q=> );
   fbAutoRise(CLK:=stCylvar.xAutoCmd , Q=> );
   fbAutoFall(CLK:=stCylvar.xAutoCmd , Q=> );
      
    //1,手动操作时，如果满足安全条件且未屏蔽了手自动不一致报警时，则输出点反转，  
    IF xReady AND (NOT xManuAlmDisable) AND fbManuFall.Q THEN
   	    xOutput  := NOT xOutput ;
		//手动操作生效时，判断输出点状态与自动命令是否一致，不一致时,置位手动操作执行中报警；一致时复位该报警。
	    //当因安全条件不满足导致自动命令未执行时，可通过手动操作控制其动作执行,此时手动操作并不引起手动操作执行中报警。
		 IF ( stCylvar.xAutoCmd ) XOR xOutput THEN
   	   	    f_xManuAlm  :=TRUE;
   	     ELSE 
   	   	    f_xManuAlm  :=FALSE;
   	     END_IF  	 	
     END_IF
	 
	//2,手动操作时，如果满足安全条件且屏蔽了手自动不一致报警时，则自动控制点反转、复位手自动不一致报警，  
    IF xReady AND  xManuAlmDisable AND fbManuFall.Q THEN
   	    stCylvar.xAutoCmd  := NOT stCylvar.xAutoCmd ;
		f_xManuAlm  :=FALSE;		  	 	
    END_IF
   
   
   
   //自动命令置位时，如果满足安全条件，则输出点置位
   IF xReady AND fbAutoRise.Q THEN
   	   xOutput  :=TRUE;
   END_IF
      
   //自动命令复位时，如满足安全条件，则输出点复位。
   IF xReady AND fbAutoFall.Q THEN
   	    xOutput  :=FALSE;		
   END_IF
   
   
   //原位状态输出
   fbBackTon(IN:= ( NOT xOutput) AND ( NOT xFrontSensor ) AND ( xBackSensor OR xBackSensorDisable ) , PT:= WORD_TO_TIME ( wBackDelay *10 ) , Q=> stCylvar.xIsBack, ET=> );
   
   
   //到位状态输出
   fbFrontTon(IN:= xOutput AND ( xFrontSensor OR xFrontSensorDisable ) AND ( NOT xBackSensor ) , PT:= WORD_TO_TIME ( wFrontDelay *10 ), Q=> stCylvar.xIsFront, ET=> );
      
	  
   //报警复位
   fbResetRise(CLK:= xReset, Q=> );
   IF fbResetRise.Q THEN
   	   f_xNotRdyAlm := FALSE;
	   f_xFrontAlm := FALSE;
	   f_xBackAlm := FALSE;
   
   END_IF
   
   
   //未满足安全条件报警
   //当手动操作或自动命令状态发生改变时，如果不能满足安全条件，则输出未满足安全条件报警
   IF ( fbManuFall.Q OR fbAutoRise.Q OR fbAutoFall.Q ) AND ( NOT xReady ) THEN
   	    f_xNotRdyAlm := TRUE; 
   END_IF
   
   
   //未在原位报警
   //自动命令变OFF后(上电后气缸处于自由状态时不判断)，延时5秒，如果原位标志未变为ON、且未发生手动操作和安全条件报警，则输出未到原位报警
   fbBackWait(IN:=  NOT stCylvar.xAutoCmd  , PT:= T#5S , Q=> , ET=> );
   fbBackFall(CLK:= stCylvar.xIsBack , Q=> );
   IF (( fbBackWait.Q AND (NOT stCylvar.xIsBack )) OR (( NOT stCylvar.xAutoCmd ) AND fbBackFall.Q )) AND  ( NOT f_xManuAlm ) AND  ( NOT f_xNotRdyAlm ) THEN
   	    f_xBackAlm := TRUE;
   END_IF
   
   
   //未到位报警
   //自动命令变ON后，延时5秒，如果到位标志未变为ON、且未发生手动操作和安全条件报警，则输出未到位报警
   fbFrontWait(IN:= stCylvar.xAutoCmd , PT:= T#5S , Q=> , ET=> );
   fbFrontFall(CLK:= stCylvar.xIsFront, Q=> );
   IF ( ( fbFrontWait.Q AND ( NOT stCylvar.xIsFront ) ) OR (stCylvar.xAutoCmd AND fbFrontFall.Q )) AND ( NOT f_xManuAlm ) AND ( NOT f_xNotRdyAlm ) THEN
   	    f_xFrontAlm := TRUE;   
   END_IF

END_FUNCTION_BLOCK

// Device/Application/FunctionBlock/Public_Prog
PROGRAM Public_Prog
VAR
	Clock_10Hz: FB102_ClockPuls;
	Clock_5Hz: FB102_ClockPuls;
	Clock_2Hz: FB102_ClockPuls;
	Clock_1Hz: FB102_ClockPuls;
	Clock_HalfHz: FB102_ClockPuls;
END_VAR
VAR // added by the converter: edge detectors and wires of the graphical bodies
    _rt1 : R_TRIG;
END_VAR

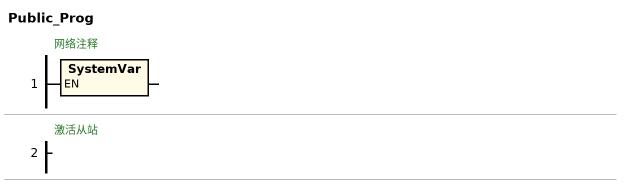
// NETWORK 1
// 网络注释
SystemVar();

// NETWORK 2
// 激活从站

ACTION SystemVar:
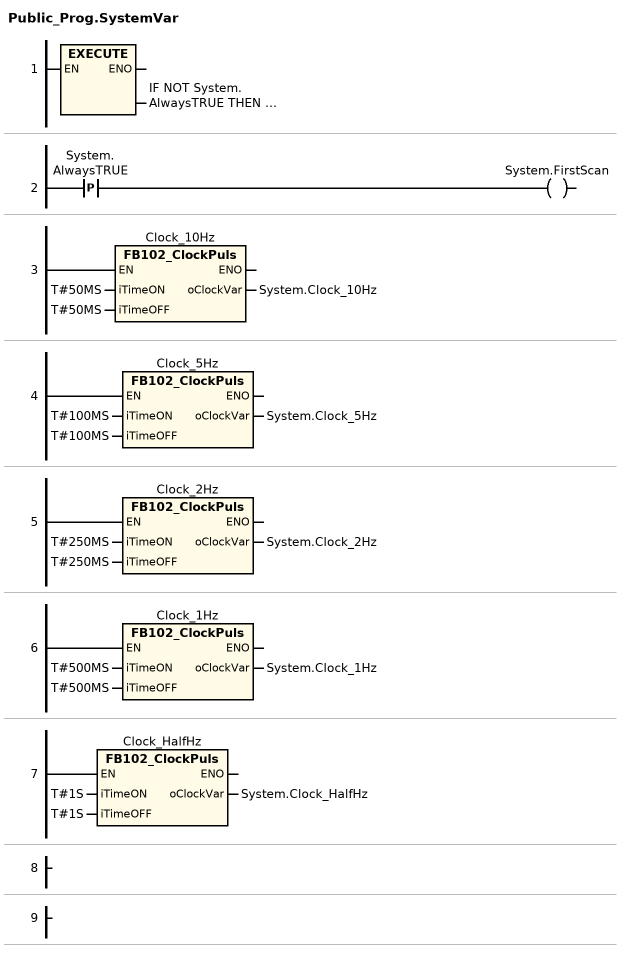
// NETWORK 1
IF NOT System.AlwaysTRUE THEN
	System.AlwaysTRUE := TRUE;
END_IF
IF  System.AlwaysFALSE THEN
	System.AlwaysFALSE := FALSE;
END_IF
IF NOT Publics.CYGIA_ON THEN
	Publics.CYGIA_ON := TRUE;
END_IF
IF  Publics.CYGIA_OFF THEN
	Publics.CYGIA_OFF := FALSE;
END_IF

// NETWORK 2
_rt1(CLK := System.AlwaysTRUE);
System.FirstScan := _rt1.Q;

// NETWORK 3
Clock_10Hz(iTimeON := T#50MS, iTimeOFF := T#50MS, oClockVar => System.Clock_10Hz); // FB102_ClockPuls

// NETWORK 4
Clock_5Hz(iTimeON := T#100MS, iTimeOFF := T#100MS, oClockVar => System.Clock_5Hz); // FB102_ClockPuls

// NETWORK 5
Clock_2Hz(iTimeON := T#250MS, iTimeOFF := T#250MS, oClockVar => System.Clock_2Hz); // FB102_ClockPuls

// NETWORK 6
Clock_1Hz(iTimeON := T#500MS, iTimeOFF := T#500MS, oClockVar => System.Clock_1Hz); // FB102_ClockPuls

// NETWORK 7
Clock_HalfHz(iTimeON := T#1S, iTimeOFF := T#1S, oClockVar => System.Clock_HalfHz); // FB102_ClockPuls

// NETWORK 8

// NETWORK 9
END_ACTION

END_PROGRAM

// Device/Application/FunctionBlock/FB102_ClockPuls
FUNCTION_BLOCK FB102_ClockPuls
VAR_INPUT
	///脉冲ON时间
	iTimeON: TIME;
	///脉冲OFF时间
	iTimeOFF: TIME;
END_VAR
VAR_OUTPUT
	///时钟脉冲差速器
	oClockVar: BOOL;
END_VAR
VAR
	TON_Clock: TON;
	TOF_Clock: TOF;
END_VAR

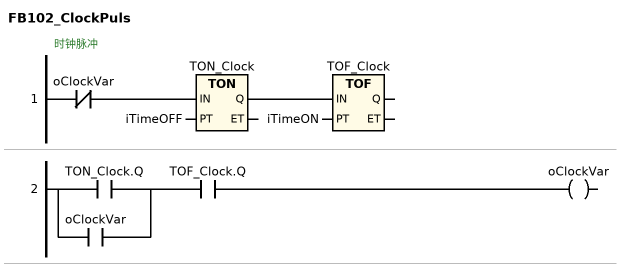
// NETWORK 1
// 时钟脉冲
TON_Clock(IN := NOT oClockVar, PT := iTimeOFF); // TON
TOF_Clock(IN := TON_Clock.Q, PT := iTimeON); // TOF

// NETWORK 2
oClockVar := (TON_Clock.Q OR oClockVar) AND TOF_Clock.Q;

END_FUNCTION_BLOCK

// Device/Application/OP1001
PROGRAM OP1001
VAR
	启动自锁: BOOL;
	下次循环: word;
	当次循环: word;
	循环停止: BOOL;
	阻止运行条件: BOOL;
	TON_0: TON;
	TON_1: TON;
	TON_2: TON;
	通知_允许抓取物料: BOOL;
	通知_物料抓取完成: BOOL;
END_VAR
VAR // added by the converter: edge detectors and wires of the graphical bodies
    _rt1 : R_TRIG;
    _w1, _w2, _w3, _w4, _w5, _w6 : BOOL;
END_VAR

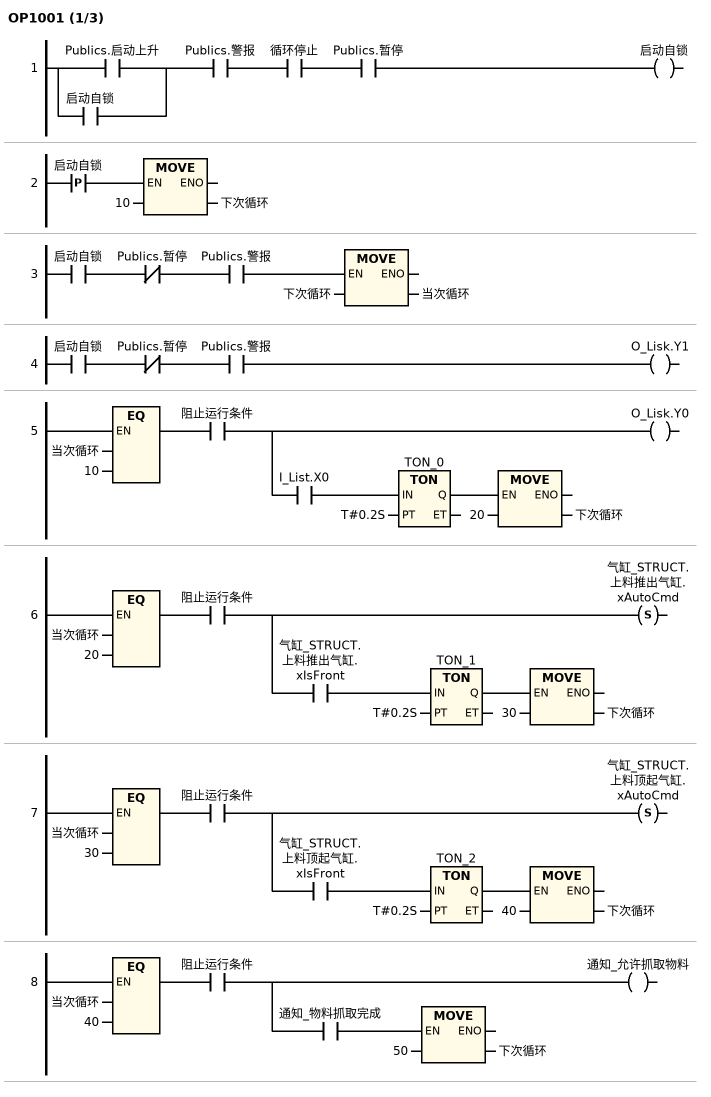
// NETWORK 1
启动自锁 := (Publics.启动上升 OR 启动自锁) AND Publics.警报 AND 循环停止 AND Publics.暂停;

// NETWORK 2
_rt1(CLK := 启动自锁);
IF _rt1.Q THEN 下次循环 := 10; END_IF

// NETWORK 3
IF 启动自锁 AND NOT Publics.暂停 AND Publics.警报 THEN 当次循环 := 下次循环; END_IF

// NETWORK 4
O_Lisk.Y1 := 启动自锁 AND NOT Publics.暂停 AND Publics.警报;

// NETWORK 5
_w1 := 当次循环 = 10 AND 阻止运行条件;
O_Lisk.Y0 := _w1;
TON_0(IN := _w1 AND I_List.X0, PT := T#0.2S); // TON
IF TON_0.Q THEN 下次循环 := 20; END_IF

// NETWORK 6
_w2 := 当次循环 = 20 AND 阻止运行条件;
气缸_STRUCT.上料推出气缸.xAutoCmd S= _w2;
TON_1(IN := _w2 AND 气缸_STRUCT.上料推出气缸.xIsFront, PT := T#0.2S); // TON
IF TON_1.Q THEN 下次循环 := 30; END_IF

// NETWORK 7
_w3 := 当次循环 = 30 AND 阻止运行条件;
气缸_STRUCT.上料顶起气缸.xAutoCmd S= _w3;
TON_2(IN := _w3 AND 气缸_STRUCT.上料顶起气缸.xIsFront, PT := T#0.2S); // TON
IF TON_2.Q THEN 下次循环 := 40; END_IF

// NETWORK 8
_w4 := 当次循环 = 40 AND 阻止运行条件;
通知_允许抓取物料 := _w4;
IF _w4 AND 通知_物料抓取完成 THEN 下次循环 := 50; END_IF

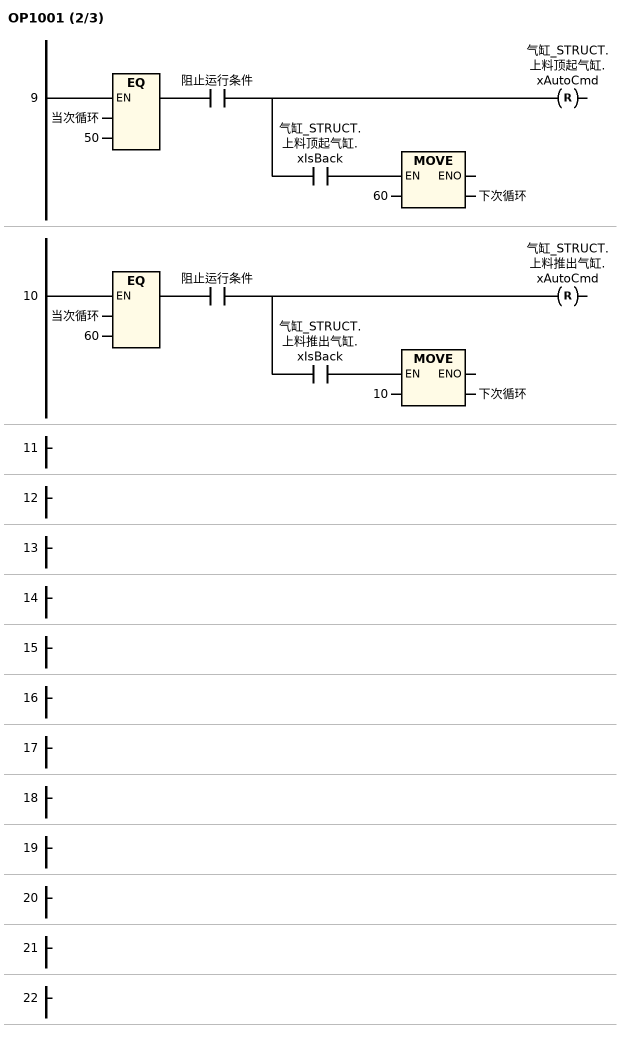
// NETWORK 9
_w5 := 当次循环 = 50 AND 阻止运行条件;
气缸_STRUCT.上料顶起气缸.xAutoCmd R= _w5;
IF _w5 AND 气缸_STRUCT.上料顶起气缸.xIsBack THEN 下次循环 := 60; END_IF

// NETWORK 10
_w6 := 当次循环 = 60 AND 阻止运行条件;
气缸_STRUCT.上料推出气缸.xAutoCmd R= _w6;
IF _w6 AND 气缸_STRUCT.上料推出气缸.xIsBack THEN 下次循环 := 10; END_IF

// NETWORK 11

// NETWORK 12

// NETWORK 13

// NETWORK 14

// NETWORK 15

// NETWORK 16

// NETWORK 17

// NETWORK 18

// NETWORK 19

// NETWORK 20

// NETWORK 21

// NETWORK 22

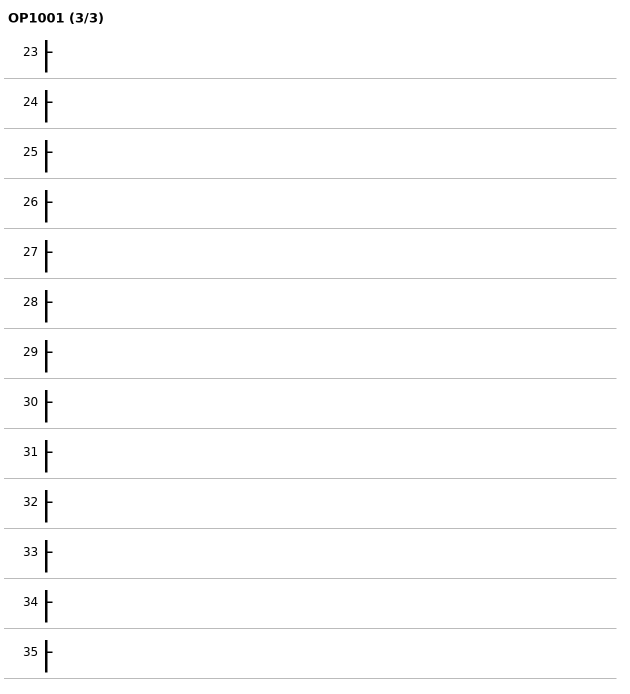
// NETWORK 23

// NETWORK 24

// NETWORK 25

// NETWORK 26

// NETWORK 27

// NETWORK 28

// NETWORK 29

// NETWORK 30

// NETWORK 31

// NETWORK 32

// NETWORK 33

// NETWORK 34

// NETWORK 35

END_PROGRAM

// Device/Application/OP1002
PROGRAM OP1002
VAR
	启动自锁: BOOL;
	循环停止: BOOL;
	下次循环: word;
	当次循环: word;
	伺服停止0: BOOL;
	避开扫描周期: BOOL;
	阻止运行条件: BOOL;
	通知_抓手上方要开门: BOOL;
	通知_门打开完成: BOOL;
	通知_关门: BOOL;
	通知_门关上了: BOOL;
	Y30_联机自锁: BOOL;
	TON_0: TON;
END_VAR
VAR // added by the converter: edge detectors and wires of the graphical bodies
    _rt1, _rt2, _rt3 : R_TRIG;
    _ft1 : F_TRIG;
    _w1, _w2, _w3, _w4, _w5, _w6, _w7, _w8, _w9, _w10, _w11, _w12, _w13, _w14, _w15, _w16, _w17, _w18, _w19, _w20, _w21, _w22, _w23, _w24, _w25, _w26, _w27, _w28, _w29, _w30, _w31, _w32, _w33, _w34, _w35, _w36, _w37, _w38, _w39, _w40, _w41, _w42, _w43, _w44, _w45, _w46, _w47, _w48, _w49, _w50, _w51, _w52, _w53, _w54, _w55, _w56, _w57, _w58, _w59 : BOOL;
END_VAR

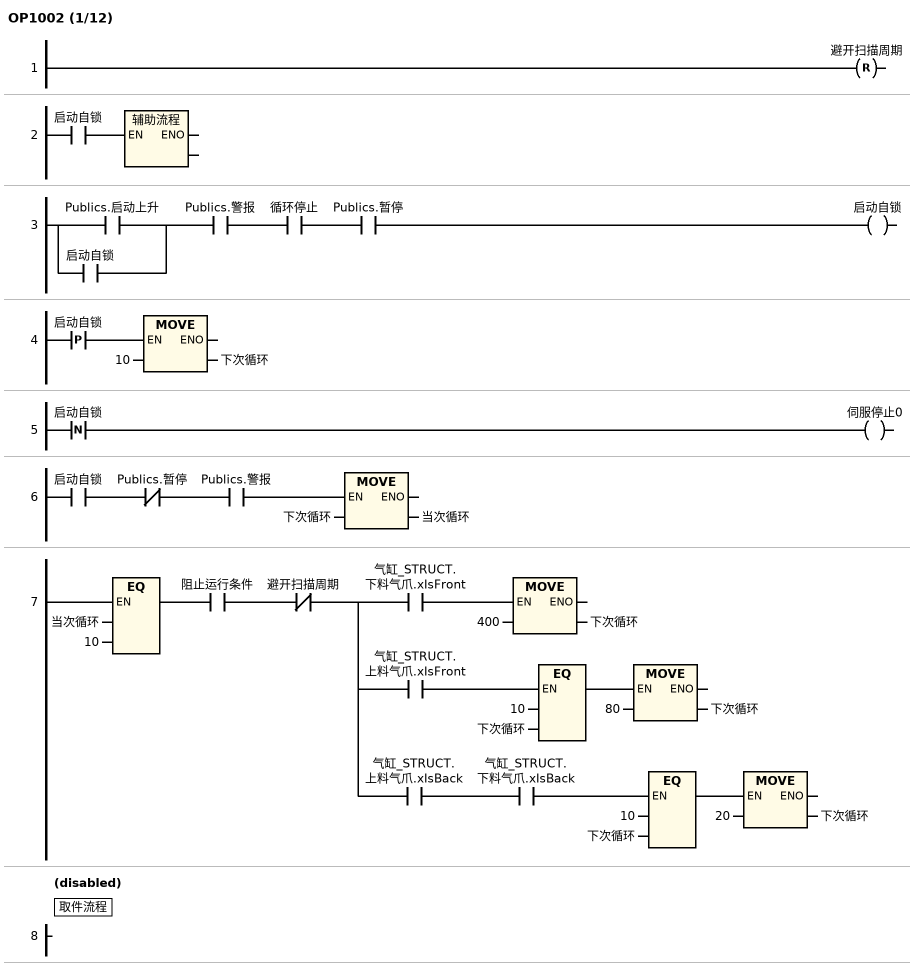
// NETWORK 1
避开扫描周期 R= TRUE;

// NETWORK 2
IF 启动自锁 THEN 辅助流程(); END_IF

// NETWORK 3
启动自锁 := (Publics.启动上升 OR 启动自锁) AND Publics.警报 AND 循环停止 AND Publics.暂停;

// NETWORK 4
_rt1(CLK := 启动自锁);
IF _rt1.Q THEN 下次循环 := 10; END_IF

// NETWORK 5
_ft1(CLK := 启动自锁);
伺服停止0 := _ft1.Q;

// NETWORK 6
IF 启动自锁 AND NOT Publics.暂停 AND Publics.警报 THEN 当次循环 := 下次循环; END_IF

// NETWORK 7
_w1 := 当次循环 = 10 AND 阻止运行条件 AND NOT 避开扫描周期;
IF _w1 AND 气缸_STRUCT.下料气爪.xIsFront THEN 下次循环 := 400; END_IF
IF _w1 AND 气缸_STRUCT.上料气爪.xIsFront AND 10 = 下次循环 THEN 下次循环 := 80; END_IF
IF _w1 AND 气缸_STRUCT.上料气爪.xIsBack AND 气缸_STRUCT.下料气爪.xIsBack AND 10 = 下次循环 THEN 下次循环 := 20; END_IF

// NETWORK 8 (disabled)
// label: 取件流程

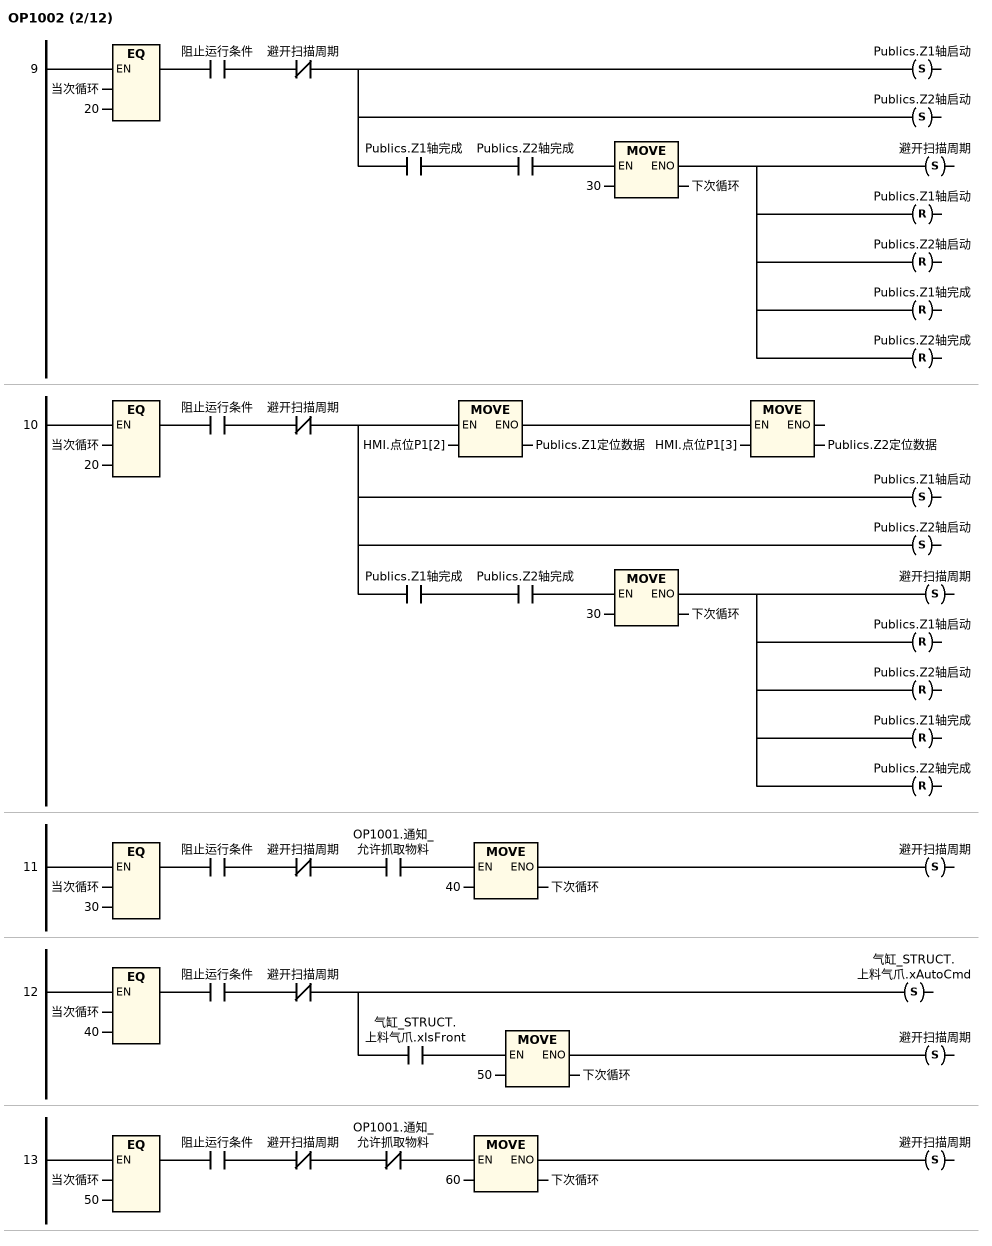
// NETWORK 9
_w2 := 当次循环 = 20 AND 阻止运行条件 AND NOT 避开扫描周期;
Publics.Z1轴启动 S= _w2;
Publics.Z2轴启动 S= _w2;
IF _w2 AND Publics.Z1轴完成 AND Publics.Z2轴完成 THEN 下次循环 := 30; END_IF
_w3 := _w2 AND Publics.Z1轴完成 AND Publics.Z2轴完成;
避开扫描周期 S= _w3;
Publics.Z1轴启动 R= _w3;
Publics.Z2轴启动 R= _w3;
Publics.Z1轴完成 R= _w3;
Publics.Z2轴完成 R= _w3;

// NETWORK 10
_w4 := 当次循环 = 20 AND 阻止运行条件 AND NOT 避开扫描周期;
IF _w4 THEN Publics.Z1定位数据 := HMI.点位P1[2]; END_IF
IF _w4 THEN Publics.Z2定位数据 := HMI.点位P1[3]; END_IF
Publics.Z1轴启动 S= _w4;
Publics.Z2轴启动 S= _w4;
IF _w4 AND Publics.Z1轴完成 AND Publics.Z2轴完成 THEN 下次循环 := 30; END_IF
_w5 := _w4 AND Publics.Z1轴完成 AND Publics.Z2轴完成;
避开扫描周期 S= _w5;
Publics.Z1轴启动 R= _w5;
Publics.Z2轴启动 R= _w5;
Publics.Z1轴完成 R= _w5;
Publics.Z2轴完成 R= _w5;

// NETWORK 11
_w6 := 当次循环 = 30 AND 阻止运行条件 AND NOT 避开扫描周期 AND OP1001.通知_允许抓取物料;
IF _w6 THEN 下次循环 := 40; END_IF
避开扫描周期 S= _w6;

// NETWORK 12
_w7 := 当次循环 = 40 AND 阻止运行条件 AND NOT 避开扫描周期;
气缸_STRUCT.上料气爪.xAutoCmd S= _w7;
IF _w7 AND 气缸_STRUCT.上料气爪.xIsFront THEN 下次循环 := 50; END_IF
避开扫描周期 S= _w7 AND 气缸_STRUCT.上料气爪.xIsFront;

// NETWORK 13
_w8 := 当次循环 = 50 AND 阻止运行条件 AND NOT 避开扫描周期 AND NOT OP1001.通知_允许抓取物料;
IF _w8 THEN 下次循环 := 60; END_IF
避开扫描周期 S= _w8;

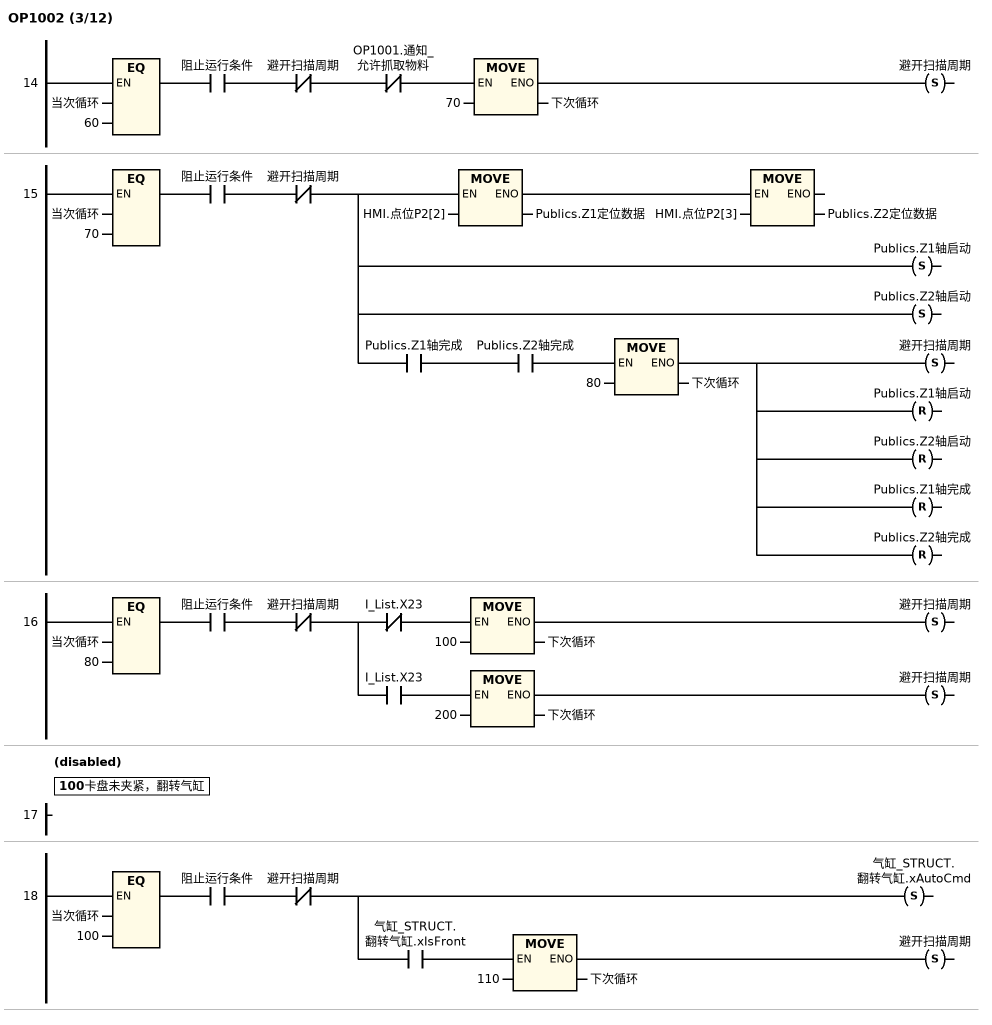
// NETWORK 14
_w9 := 当次循环 = 60 AND 阻止运行条件 AND NOT 避开扫描周期 AND NOT OP1001.通知_允许抓取物料;
IF _w9 THEN 下次循环 := 70; END_IF
避开扫描周期 S= _w9;

// NETWORK 15
_w10 := 当次循环 = 70 AND 阻止运行条件 AND NOT 避开扫描周期;
IF _w10 THEN Publics.Z1定位数据 := HMI.点位P2[2]; END_IF
IF _w10 THEN Publics.Z2定位数据 := HMI.点位P2[3]; END_IF
Publics.Z1轴启动 S= _w10;
Publics.Z2轴启动 S= _w10;
IF _w10 AND Publics.Z1轴完成 AND Publics.Z2轴完成 THEN 下次循环 := 80; END_IF
_w11 := _w10 AND Publics.Z1轴完成 AND Publics.Z2轴完成;
避开扫描周期 S= _w11;
Publics.Z1轴启动 R= _w11;
Publics.Z2轴启动 R= _w11;
Publics.Z1轴完成 R= _w11;
Publics.Z2轴完成 R= _w11;

// NETWORK 16
_w12 := 当次循环 = 80 AND 阻止运行条件 AND NOT 避开扫描周期;
IF _w12 AND NOT I_List.X23 THEN 下次循环 := 100; END_IF
避开扫描周期 S= _w12 AND NOT I_List.X23;
IF _w12 AND I_List.X23 THEN 下次循环 := 200; END_IF
避开扫描周期 S= _w12 AND I_List.X23;

// NETWORK 17 (disabled)
// label: 100卡盘未夹紧，翻转气缸

// NETWORK 18
_w13 := 当次循环 = 100 AND 阻止运行条件 AND NOT 避开扫描周期;
气缸_STRUCT.翻转气缸.xAutoCmd S= _w13;
IF _w13 AND 气缸_STRUCT.翻转气缸.xIsFront THEN 下次循环 := 110; END_IF
避开扫描周期 S= _w13 AND 气缸_STRUCT.翻转气缸.xIsFront;

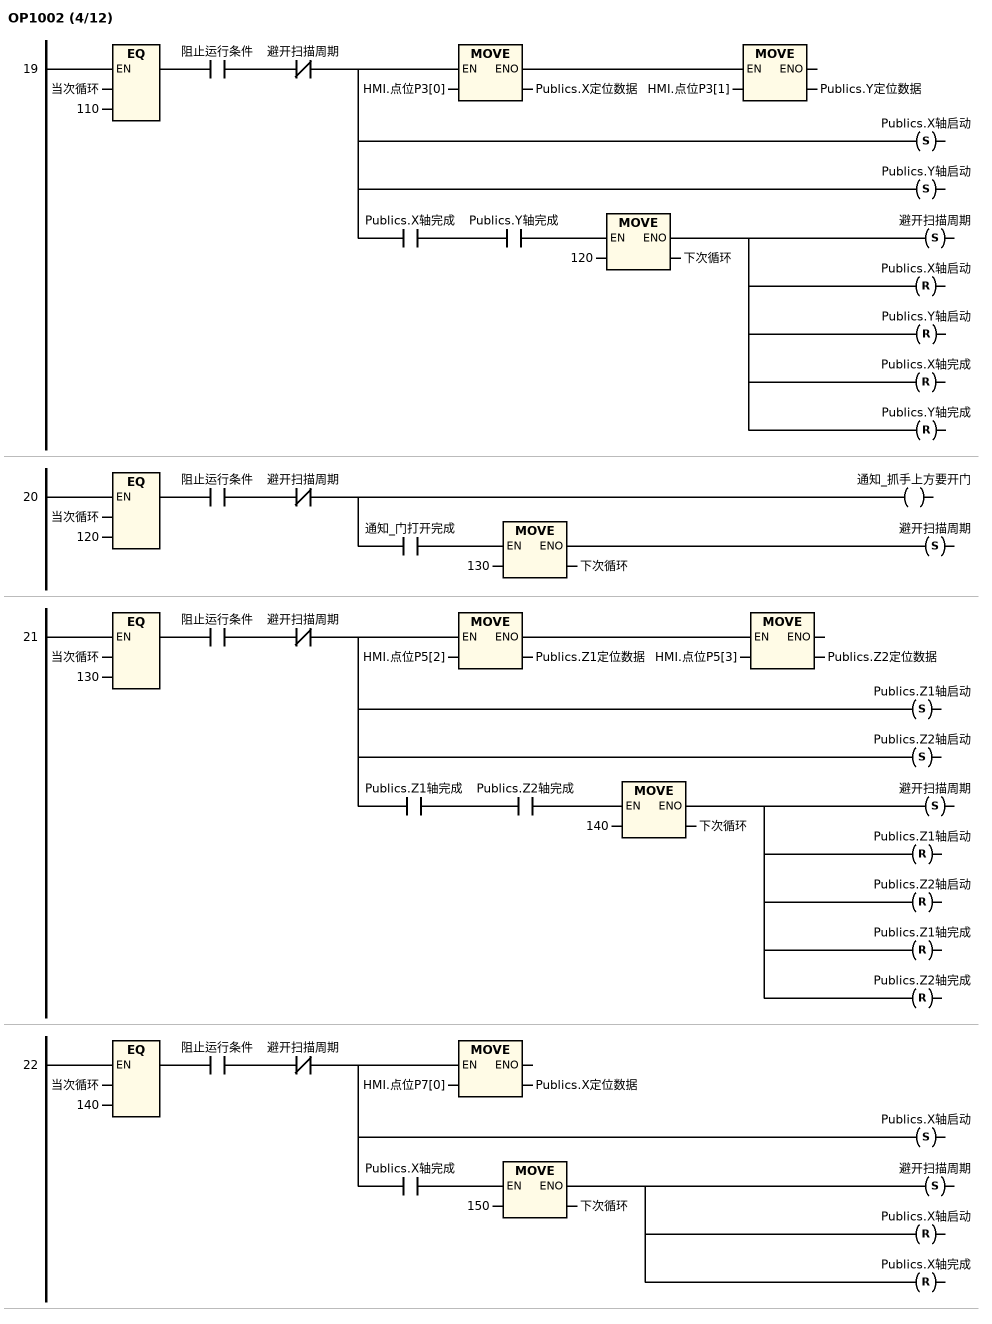
// NETWORK 19
_w14 := 当次循环 = 110 AND 阻止运行条件 AND NOT 避开扫描周期;
IF _w14 THEN Publics.X定位数据 := HMI.点位P3[0]; END_IF
IF _w14 THEN Publics.Y定位数据 := HMI.点位P3[1]; END_IF
Publics.X轴启动 S= _w14;
Publics.Y轴启动 S= _w14;
IF _w14 AND Publics.X轴完成 AND Publics.Y轴完成 THEN 下次循环 := 120; END_IF
_w15 := _w14 AND Publics.X轴完成 AND Publics.Y轴完成;
避开扫描周期 S= _w15;
Publics.X轴启动 R= _w15;
Publics.Y轴启动 R= _w15;
Publics.X轴完成 R= _w15;
Publics.Y轴完成 R= _w15;

// NETWORK 20
_w16 := 当次循环 = 120 AND 阻止运行条件 AND NOT 避开扫描周期;
通知_抓手上方要开门 := _w16;
IF _w16 AND 通知_门打开完成 THEN 下次循环 := 130; END_IF
避开扫描周期 S= _w16 AND 通知_门打开完成;

// NETWORK 21
_w17 := 当次循环 = 130 AND 阻止运行条件 AND NOT 避开扫描周期;
IF _w17 THEN Publics.Z1定位数据 := HMI.点位P5[2]; END_IF
IF _w17 THEN Publics.Z2定位数据 := HMI.点位P5[3]; END_IF
Publics.Z1轴启动 S= _w17;
Publics.Z2轴启动 S= _w17;
IF _w17 AND Publics.Z1轴完成 AND Publics.Z2轴完成 THEN 下次循环 := 140; END_IF
_w18 := _w17 AND Publics.Z1轴完成 AND Publics.Z2轴完成;
避开扫描周期 S= _w18;
Publics.Z1轴启动 R= _w18;
Publics.Z2轴启动 R= _w18;
Publics.Z1轴完成 R= _w18;
Publics.Z2轴完成 R= _w18;

// NETWORK 22
_w19 := 当次循环 = 140 AND 阻止运行条件 AND NOT 避开扫描周期;
IF _w19 THEN Publics.X定位数据 := HMI.点位P7[0]; END_IF
Publics.X轴启动 S= _w19;
IF _w19 AND Publics.X轴完成 THEN 下次循环 := 150; END_IF
_w20 := _w19 AND Publics.X轴完成;
避开扫描周期 S= _w20;
Publics.X轴启动 R= _w20;
Publics.X轴完成 R= _w20;

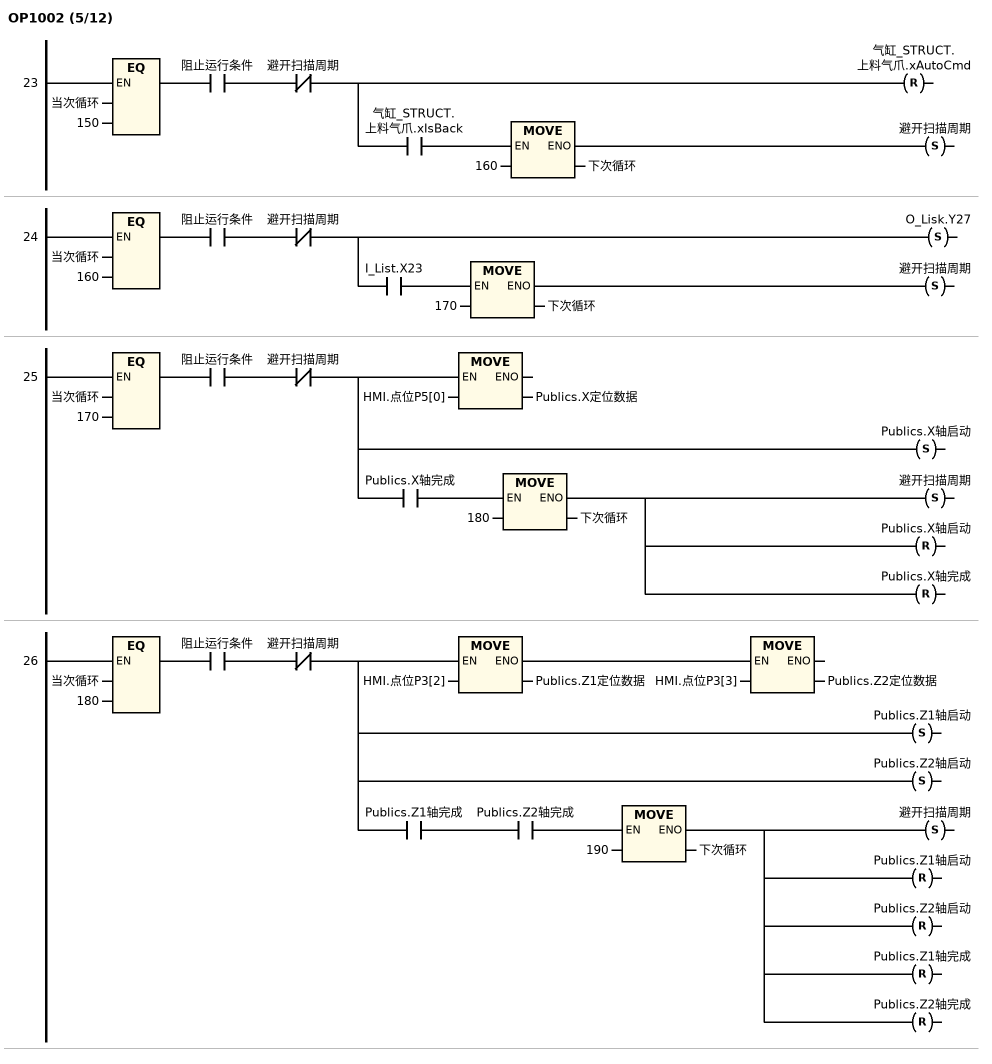
// NETWORK 23
_w21 := 当次循环 = 150 AND 阻止运行条件 AND NOT 避开扫描周期;
气缸_STRUCT.上料气爪.xAutoCmd R= _w21;
IF _w21 AND 气缸_STRUCT.上料气爪.xIsBack THEN 下次循环 := 160; END_IF
避开扫描周期 S= _w21 AND 气缸_STRUCT.上料气爪.xIsBack;

// NETWORK 24
_w22 := 当次循环 = 160 AND 阻止运行条件 AND NOT 避开扫描周期;
O_Lisk.Y27 S= _w22;
IF _w22 AND I_List.X23 THEN 下次循环 := 170; END_IF
避开扫描周期 S= _w22 AND I_List.X23;

// NETWORK 25
_w23 := 当次循环 = 170 AND 阻止运行条件 AND NOT 避开扫描周期;
IF _w23 THEN Publics.X定位数据 := HMI.点位P5[0]; END_IF
Publics.X轴启动 S= _w23;
IF _w23 AND Publics.X轴完成 THEN 下次循环 := 180; END_IF
_w24 := _w23 AND Publics.X轴完成;
避开扫描周期 S= _w24;
Publics.X轴启动 R= _w24;
Publics.X轴完成 R= _w24;

// NETWORK 26
_w25 := 当次循环 = 180 AND 阻止运行条件 AND NOT 避开扫描周期;
IF _w25 THEN Publics.Z1定位数据 := HMI.点位P3[2]; END_IF
IF _w25 THEN Publics.Z2定位数据 := HMI.点位P3[3]; END_IF
Publics.Z1轴启动 S= _w25;
Publics.Z2轴启动 S= _w25;
IF _w25 AND Publics.Z1轴完成 AND Publics.Z2轴完成 THEN 下次循环 := 190; END_IF
_w26 := _w25 AND Publics.Z1轴完成 AND Publics.Z2轴完成;
避开扫描周期 S= _w26;
Publics.Z1轴启动 R= _w26;
Publics.Z2轴启动 R= _w26;
Publics.Z1轴完成 R= _w26;
Publics.Z2轴完成 R= _w26;

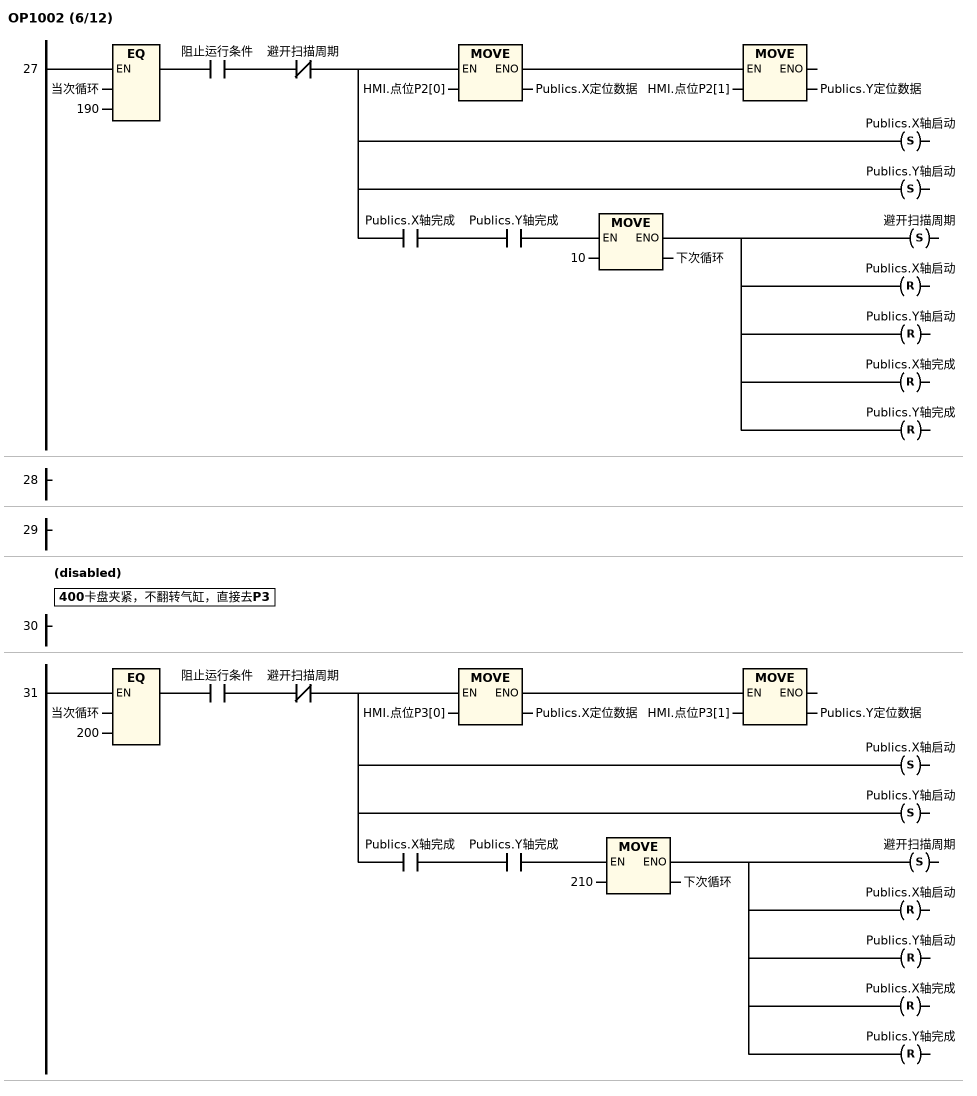
// NETWORK 27
_w27 := 当次循环 = 190 AND 阻止运行条件 AND NOT 避开扫描周期;
IF _w27 THEN Publics.X定位数据 := HMI.点位P2[0]; END_IF
IF _w27 THEN Publics.Y定位数据 := HMI.点位P2[1]; END_IF
Publics.X轴启动 S= _w27;
Publics.Y轴启动 S= _w27;
IF _w27 AND Publics.X轴完成 AND Publics.Y轴完成 THEN 下次循环 := 10; END_IF
_w28 := _w27 AND Publics.X轴完成 AND Publics.Y轴完成;
避开扫描周期 S= _w28;
Publics.X轴启动 R= _w28;
Publics.Y轴启动 R= _w28;
Publics.X轴完成 R= _w28;
Publics.Y轴完成 R= _w28;

// NETWORK 28

// NETWORK 29

// NETWORK 30 (disabled)
// label: 400卡盘夹紧，不翻转气缸，直接去P3

// NETWORK 31
_w29 := 当次循环 = 200 AND 阻止运行条件 AND NOT 避开扫描周期;
IF _w29 THEN Publics.X定位数据 := HMI.点位P3[0]; END_IF
IF _w29 THEN Publics.Y定位数据 := HMI.点位P3[1]; END_IF
Publics.X轴启动 S= _w29;
Publics.Y轴启动 S= _w29;
IF _w29 AND Publics.X轴完成 AND Publics.Y轴完成 THEN 下次循环 := 210; END_IF
_w30 := _w29 AND Publics.X轴完成 AND Publics.Y轴完成;
避开扫描周期 S= _w30;
Publics.X轴启动 R= _w30;
Publics.Y轴启动 R= _w30;
Publics.X轴完成 R= _w30;
Publics.Y轴完成 R= _w30;

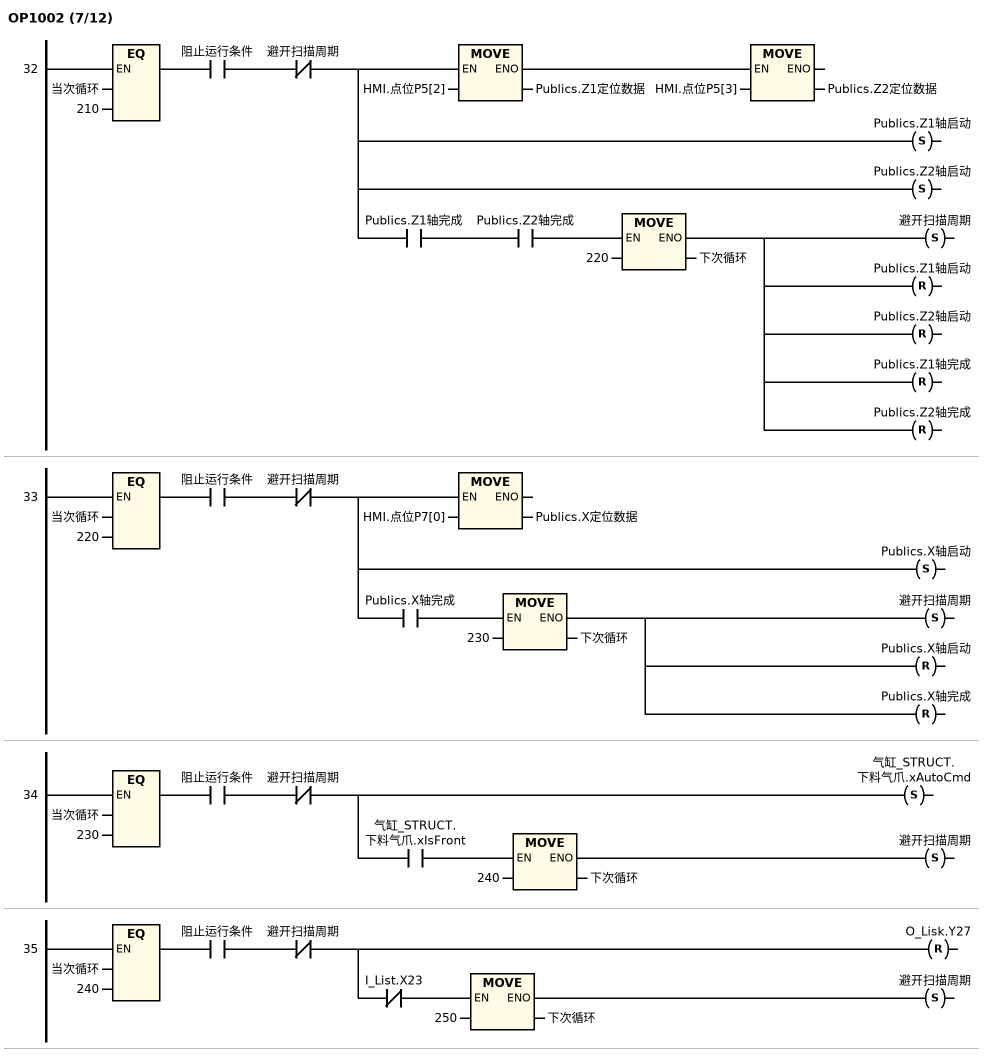
// NETWORK 32
_w31 := 当次循环 = 210 AND 阻止运行条件 AND NOT 避开扫描周期;
IF _w31 THEN Publics.Z1定位数据 := HMI.点位P5[2]; END_IF
IF _w31 THEN Publics.Z2定位数据 := HMI.点位P5[3]; END_IF
Publics.Z1轴启动 S= _w31;
Publics.Z2轴启动 S= _w31;
IF _w31 AND Publics.Z1轴完成 AND Publics.Z2轴完成 THEN 下次循环 := 220; END_IF
_w32 := _w31 AND Publics.Z1轴完成 AND Publics.Z2轴完成;
避开扫描周期 S= _w32;
Publics.Z1轴启动 R= _w32;
Publics.Z2轴启动 R= _w32;
Publics.Z1轴完成 R= _w32;
Publics.Z2轴完成 R= _w32;

// NETWORK 33
_w33 := 当次循环 = 220 AND 阻止运行条件 AND NOT 避开扫描周期;
IF _w33 THEN Publics.X定位数据 := HMI.点位P7[0]; END_IF
Publics.X轴启动 S= _w33;
IF _w33 AND Publics.X轴完成 THEN 下次循环 := 230; END_IF
_w34 := _w33 AND Publics.X轴完成;
避开扫描周期 S= _w34;
Publics.X轴启动 R= _w34;
Publics.X轴完成 R= _w34;

// NETWORK 34
_w35 := 当次循环 = 230 AND 阻止运行条件 AND NOT 避开扫描周期;
气缸_STRUCT.下料气爪.xAutoCmd S= _w35;
IF _w35 AND 气缸_STRUCT.下料气爪.xIsFront THEN 下次循环 := 240; END_IF
避开扫描周期 S= _w35 AND 气缸_STRUCT.下料气爪.xIsFront;

// NETWORK 35
_w36 := 当次循环 = 240 AND 阻止运行条件 AND NOT 避开扫描周期;
O_Lisk.Y27 R= _w36;
IF _w36 AND NOT I_List.X23 THEN 下次循环 := 250; END_IF
避开扫描周期 S= _w36 AND NOT I_List.X23;

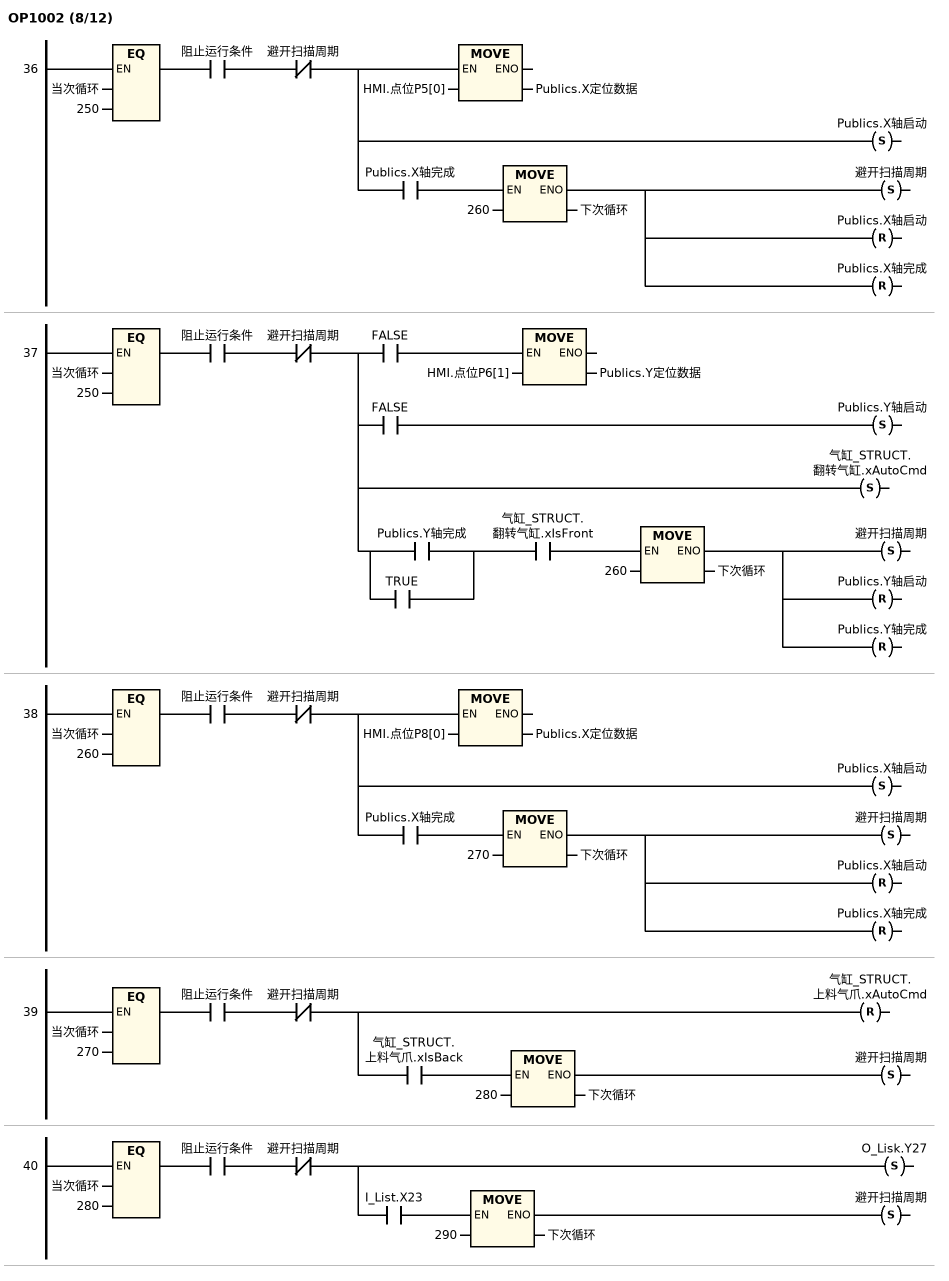
// NETWORK 36
_w37 := 当次循环 = 250 AND 阻止运行条件 AND NOT 避开扫描周期;
IF _w37 THEN Publics.X定位数据 := HMI.点位P5[0]; END_IF
Publics.X轴启动 S= _w37;
IF _w37 AND Publics.X轴完成 THEN 下次循环 := 260; END_IF
_w38 := _w37 AND Publics.X轴完成;
避开扫描周期 S= _w38;
Publics.X轴启动 R= _w38;
Publics.X轴完成 R= _w38;

// NETWORK 37
_w39 := 当次循环 = 250 AND 阻止运行条件 AND NOT 避开扫描周期;
IF _w39 AND FALSE THEN Publics.Y定位数据 := HMI.点位P6[1]; END_IF
Publics.Y轴启动 S= _w39 AND FALSE;
气缸_STRUCT.翻转气缸.xAutoCmd S= _w39;
IF _w39 AND (Publics.Y轴完成 OR TRUE) AND 气缸_STRUCT.翻转气缸.xIsFront THEN 下次循环 := 260; END_IF
_w40 := _w39 AND (Publics.Y轴完成 OR TRUE) AND 气缸_STRUCT.翻转气缸.xIsFront;
避开扫描周期 S= _w40;
Publics.Y轴启动 R= _w40;
Publics.Y轴完成 R= _w40;

// NETWORK 38
_w41 := 当次循环 = 260 AND 阻止运行条件 AND NOT 避开扫描周期;
IF _w41 THEN Publics.X定位数据 := HMI.点位P8[0]; END_IF
Publics.X轴启动 S= _w41;
IF _w41 AND Publics.X轴完成 THEN 下次循环 := 270; END_IF
_w42 := _w41 AND Publics.X轴完成;
避开扫描周期 S= _w42;
Publics.X轴启动 R= _w42;
Publics.X轴完成 R= _w42;

// NETWORK 39
_w43 := 当次循环 = 270 AND 阻止运行条件 AND NOT 避开扫描周期;
气缸_STRUCT.上料气爪.xAutoCmd R= _w43;
IF _w43 AND 气缸_STRUCT.上料气爪.xIsBack THEN 下次循环 := 280; END_IF
避开扫描周期 S= _w43 AND 气缸_STRUCT.上料气爪.xIsBack;

// NETWORK 40
_w44 := 当次循环 = 280 AND 阻止运行条件 AND NOT 避开扫描周期;
O_Lisk.Y27 S= _w44;
IF _w44 AND I_List.X23 THEN 下次循环 := 290; END_IF
避开扫描周期 S= _w44 AND I_List.X23;

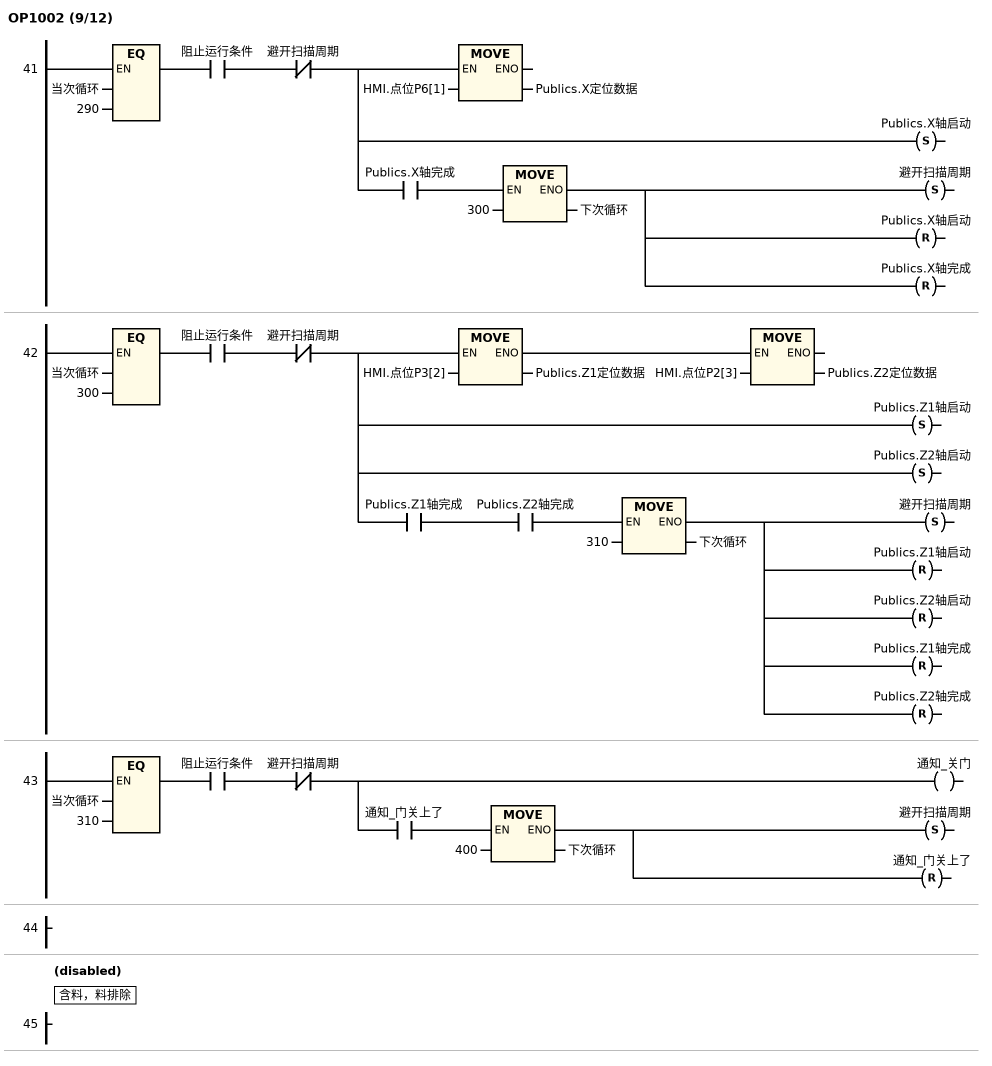
// NETWORK 41
_w45 := 当次循环 = 290 AND 阻止运行条件 AND NOT 避开扫描周期;
IF _w45 THEN Publics.X定位数据 := HMI.点位P6[1]; END_IF
Publics.X轴启动 S= _w45;
IF _w45 AND Publics.X轴完成 THEN 下次循环 := 300; END_IF
_w46 := _w45 AND Publics.X轴完成;
避开扫描周期 S= _w46;
Publics.X轴启动 R= _w46;
Publics.X轴完成 R= _w46;

// NETWORK 42
_w47 := 当次循环 = 300 AND 阻止运行条件 AND NOT 避开扫描周期;
IF _w47 THEN Publics.Z1定位数据 := HMI.点位P3[2]; END_IF
IF _w47 THEN Publics.Z2定位数据 := HMI.点位P2[3]; END_IF
Publics.Z1轴启动 S= _w47;
Publics.Z2轴启动 S= _w47;
IF _w47 AND Publics.Z1轴完成 AND Publics.Z2轴完成 THEN 下次循环 := 310; END_IF
_w48 := _w47 AND Publics.Z1轴完成 AND Publics.Z2轴完成;
避开扫描周期 S= _w48;
Publics.Z1轴启动 R= _w48;
Publics.Z2轴启动 R= _w48;
Publics.Z1轴完成 R= _w48;
Publics.Z2轴完成 R= _w48;

// NETWORK 43
_w49 := 当次循环 = 310 AND 阻止运行条件 AND NOT 避开扫描周期;
通知_关门 := _w49;
IF _w49 AND 通知_门关上了 THEN 下次循环 := 400; END_IF
_w50 := _w49 AND 通知_门关上了;
避开扫描周期 S= _w50;
通知_门关上了 R= _w50;

// NETWORK 44

// NETWORK 45 (disabled)
// label: 含料，料排除

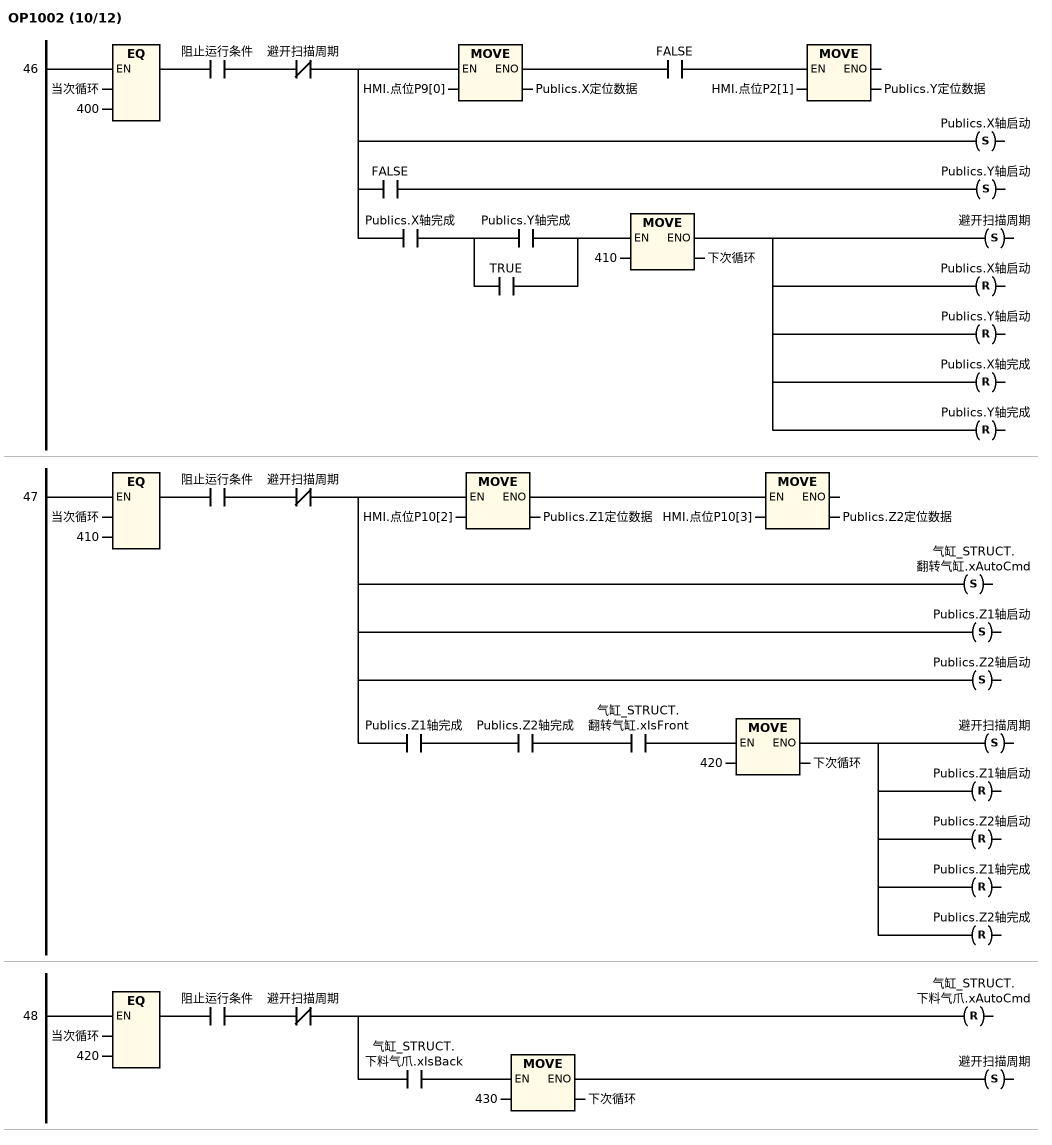
// NETWORK 46
_w51 := 当次循环 = 400 AND 阻止运行条件 AND NOT 避开扫描周期;
IF _w51 THEN Publics.X定位数据 := HMI.点位P9[0]; END_IF
IF _w51 AND FALSE THEN Publics.Y定位数据 := HMI.点位P2[1]; END_IF
Publics.X轴启动 S= _w51;
Publics.Y轴启动 S= _w51 AND FALSE;
IF _w51 AND Publics.X轴完成 AND (Publics.Y轴完成 OR TRUE) THEN 下次循环 := 410; END_IF
_w52 := _w51 AND Publics.X轴完成 AND (Publics.Y轴完成 OR TRUE);
避开扫描周期 S= _w52;
Publics.X轴启动 R= _w52;
Publics.Y轴启动 R= _w52;
Publics.X轴完成 R= _w52;
Publics.Y轴完成 R= _w52;

// NETWORK 47
_w53 := 当次循环 = 410 AND 阻止运行条件 AND NOT 避开扫描周期;
IF _w53 THEN Publics.Z1定位数据 := HMI.点位P10[2]; END_IF
IF _w53 THEN Publics.Z2定位数据 := HMI.点位P10[3]; END_IF
气缸_STRUCT.翻转气缸.xAutoCmd S= _w53;
Publics.Z1轴启动 S= _w53;
Publics.Z2轴启动 S= _w53;
IF _w53 AND Publics.Z1轴完成 AND Publics.Z2轴完成 AND 气缸_STRUCT.翻转气缸.xIsFront THEN 下次循环 := 420; END_IF
_w54 := _w53 AND Publics.Z1轴完成 AND Publics.Z2轴完成 AND 气缸_STRUCT.翻转气缸.xIsFront;
避开扫描周期 S= _w54;
Publics.Z1轴启动 R= _w54;
Publics.Z2轴启动 R= _w54;
Publics.Z1轴完成 R= _w54;
Publics.Z2轴完成 R= _w54;

// NETWORK 48
_w55 := 当次循环 = 420 AND 阻止运行条件 AND NOT 避开扫描周期;
气缸_STRUCT.下料气爪.xAutoCmd R= _w55;
IF _w55 AND 气缸_STRUCT.下料气爪.xIsBack THEN 下次循环 := 430; END_IF
避开扫描周期 S= _w55 AND 气缸_STRUCT.下料气爪.xIsBack;

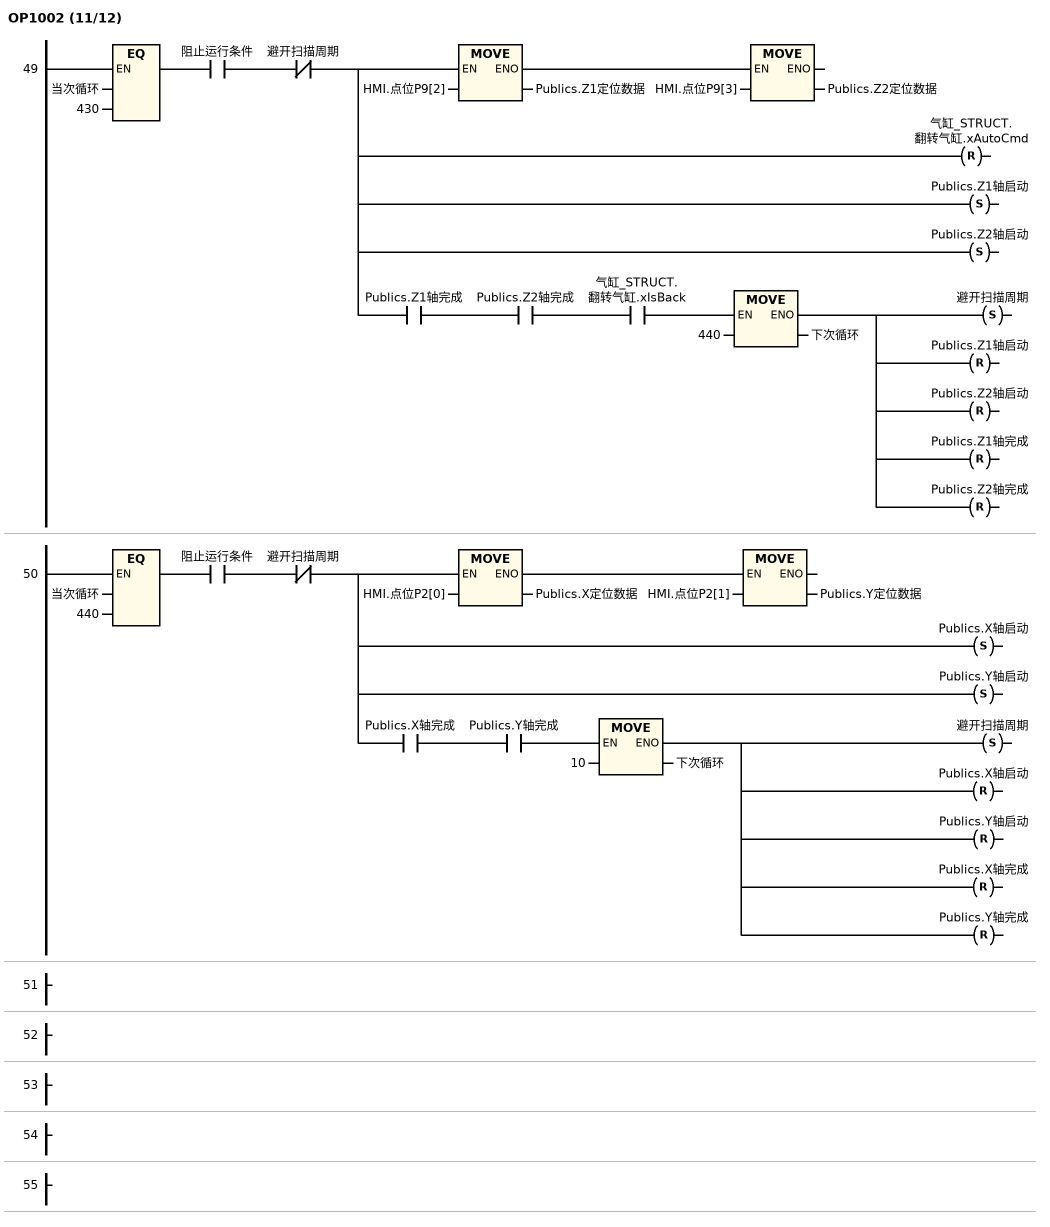
// NETWORK 49
_w56 := 当次循环 = 430 AND 阻止运行条件 AND NOT 避开扫描周期;
IF _w56 THEN Publics.Z1定位数据 := HMI.点位P9[2]; END_IF
IF _w56 THEN Publics.Z2定位数据 := HMI.点位P9[3]; END_IF
气缸_STRUCT.翻转气缸.xAutoCmd R= _w56;
Publics.Z1轴启动 S= _w56;
Publics.Z2轴启动 S= _w56;
IF _w56 AND Publics.Z1轴完成 AND Publics.Z2轴完成 AND 气缸_STRUCT.翻转气缸.xIsBack THEN 下次循环 := 440; END_IF
_w57 := _w56 AND Publics.Z1轴完成 AND Publics.Z2轴完成 AND 气缸_STRUCT.翻转气缸.xIsBack;
避开扫描周期 S= _w57;
Publics.Z1轴启动 R= _w57;
Publics.Z2轴启动 R= _w57;
Publics.Z1轴完成 R= _w57;
Publics.Z2轴完成 R= _w57;

// NETWORK 50
_w58 := 当次循环 = 440 AND 阻止运行条件 AND NOT 避开扫描周期;
IF _w58 THEN Publics.X定位数据 := HMI.点位P2[0]; END_IF
IF _w58 THEN Publics.Y定位数据 := HMI.点位P2[1]; END_IF
Publics.X轴启动 S= _w58;
Publics.Y轴启动 S= _w58;
IF _w58 AND Publics.X轴完成 AND Publics.Y轴完成 THEN 下次循环 := 10; END_IF
_w59 := _w58 AND Publics.X轴完成 AND Publics.Y轴完成;
避开扫描周期 S= _w59;
Publics.X轴启动 R= _w59;
Publics.Y轴启动 R= _w59;
Publics.X轴完成 R= _w59;
Publics.Y轴完成 R= _w59;

// NETWORK 51

// NETWORK 52

// NETWORK 53

// NETWORK 54

// NETWORK 55

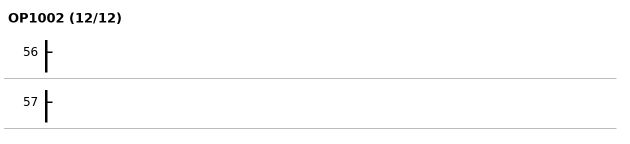
// NETWORK 56

// NETWORK 57

ACTION 辅助流程:
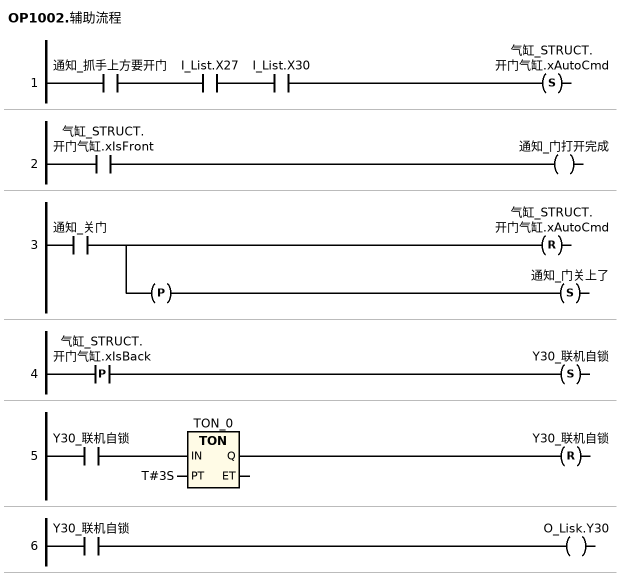
// NETWORK 1
气缸_STRUCT.开门气缸.xAutoCmd S= 通知_抓手上方要开门 AND I_List.X27 AND I_List.X30;

// NETWORK 2
通知_门打开完成 := 气缸_STRUCT.开门气缸.xIsFront;

// NETWORK 3
气缸_STRUCT.开门气缸.xAutoCmd R= 通知_关门;
_rt2(CLK := 通知_关门);
通知_门关上了 S= _rt2.Q;

// NETWORK 4
_rt3(CLK := 气缸_STRUCT.开门气缸.xIsBack);
Y30_联机自锁 S= _rt3.Q;

// NETWORK 5
TON_0(IN := Y30_联机自锁, PT := T#3S); // TON
Y30_联机自锁 R= TON_0.Q;

// NETWORK 6
O_Lisk.Y30 := Y30_联机自锁;
END_ACTION

END_PROGRAM

// Device/Application/Servo_Ctrol
PROGRAM Servo_Ctrol
VAR
	总线复位: BOOL;
	SMC3_ReinitDrive_0: SMC3_ReinitDrive;
	SMC3_ReinitDrive_1: SMC3_ReinitDrive;
	SMC3_ReinitDrive_2: SMC3_ReinitDrive;
	SMC3_ReinitDrive_3: SMC3_ReinitDrive;
	Y轴_使能: MC_Power;
	Z2轴_使能: MC_Power;
	Z1轴_使能: MC_Power;
	X轴_使能: MC_Power;
	MC_Jog_0: MC_Jog;
	Y轴_JOG: MC_Jog;
	Z2轴_JOG: MC_Jog;
	Z1轴_JOG: MC_Jog;
	X轴_JOG: MC_Jog;
	AXIS3: AXIS_REF_SM3;
	MC_Reset_0: MC_Reset;
	MC_Reset_1: MC_Reset;
	MC_Reset_2: MC_Reset;
	MC_Reset_3: MC_Reset;
	MC_ReadStatus_0: MC_ReadStatus;
	MC_ReadAxisError_0: MC_ReadAxisError;
	MC_ReadActualPosition_0: MC_ReadActualPosition;
	MC_ReadActualPosition_1: MC_ReadActualPosition;
	MC_ReadActualPosition_2: MC_ReadActualPosition;
	MC_ReadActualPosition_3: MC_ReadActualPosition;
	MC_Halt_0: MC_Halt;
	MC_Halt_1: MC_Halt;
	MC_Halt_2: MC_Halt;
	MC_Halt_3: MC_Halt;
	MC_Stop_0: MC_Stop;
	MC_Stop_1: MC_Stop;
	MC_Stop_2: MC_Stop;
	MC_Stop_3: MC_Stop;
	Z2定位: MC_MoveAbsolute;
	Z1定位: MC_MoveAbsolute;
	Y定位: MC_MoveAbsolute;
	X定位: MC_MoveAbsolute;
END_VAR
VAR // added by the converter: edge detectors and wires of the graphical bodies
    _rt1, _rt2, _rt3, _rt4, _rt5, _rt6, _rt7 : R_TRIG;
END_VAR

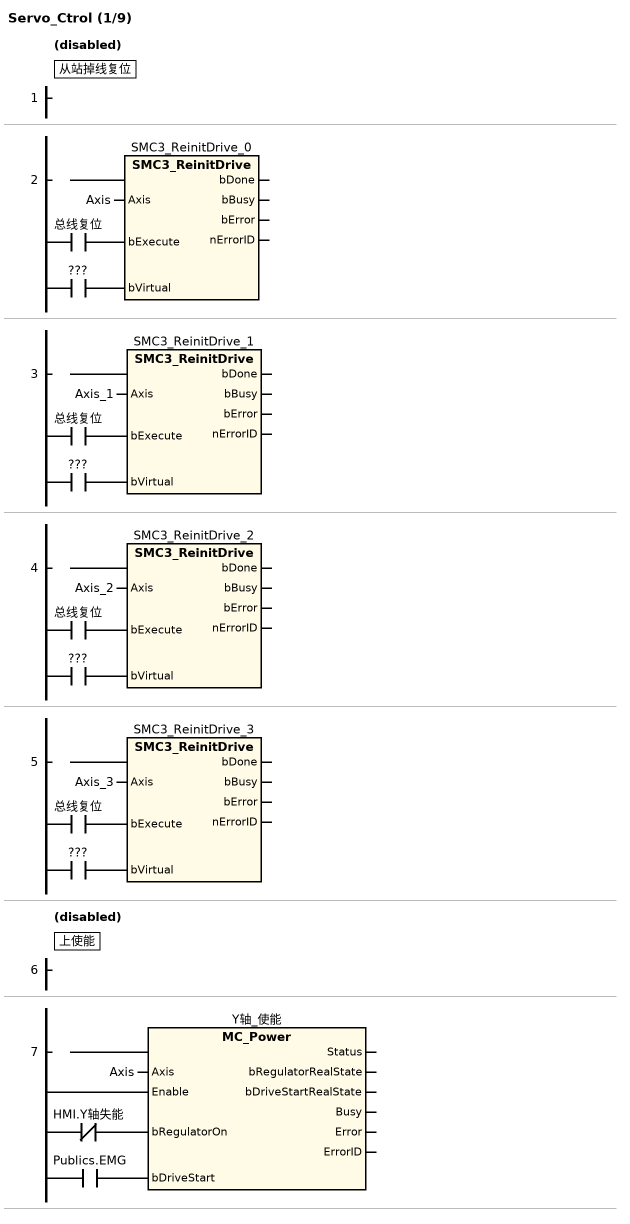
// NETWORK 1 (disabled)
// label: 从站掉线复位

// NETWORK 2
SMC3_ReinitDrive_0(Axis := Axis, bExecute := 总线复位); // SMC3_ReinitDrive

// NETWORK 3
SMC3_ReinitDrive_1(Axis := Axis_1, bExecute := 总线复位); // SMC3_ReinitDrive

// NETWORK 4
SMC3_ReinitDrive_2(Axis := Axis_2, bExecute := 总线复位); // SMC3_ReinitDrive

// NETWORK 5
SMC3_ReinitDrive_3(Axis := Axis_3, bExecute := 总线复位); // SMC3_ReinitDrive

// NETWORK 6 (disabled)
// label: 上使能

// NETWORK 7
Y轴_使能(Axis := Axis, Enable := TRUE, bRegulatorOn := NOT HMI.Y轴失能, bDriveStart := Publics.EMG); // MC_Power

